// TIA Portal V18 export
// export: Created 2025-12-01T12:38:16.9632914Z, ExportSetting None, DisplayName Totally Integrated Automation Portal, DisplayVersion V18 Update 5, DisplayName TIA Portal Openness, DisplayVersion V18 Update 5, DisplayName TIA Portal Teamcenter Gateway, DisplayVersion V18, DisplayName TIA Portal Version Control Interface, DisplayVersion V18, DisplayName STEP 7 Professional, DisplayVersion V18 Update 5, DisplayName STEP 7 Safety, DisplayVersion V18, DisplayName WinCC Professional, DisplayVersion V18 Update 5
FUNCTION_BLOCK "ST10_Flow15_FRobot_3"   // FB1085, GRAPH
// stored: AcknowledgeErrorsRequired false, AutoNumber false, GraphVersion 6.0, InitialValuesAcquisition false, SetENOAutomatically false
   // inherited from GRAPH_BASE
   VAR_INPUT
      iSysInface : "RCS_SysComInterface_V1";
   END_VAR
   VAR_IN_OUT
      ioPM_Inface : "RCS_PMInterface_V1";
      ioStatus : Int;
   END_VAR
   VAR
      sCtrlMode { S7_SetPoint := 'True'} : "SysFlowCtrlGraph";
      sUpdMES_Data : Bool;   // 更新MES数据
      工件放行中 : Bool;
      前站站号 { ExternalAccessible := 'False'; ExternalVisible := 'False'; ExternalWritable := 'False'} : UInt;
      本站站号 { ExternalAccessible := 'False'; ExternalVisible := 'False'; ExternalWritable := 'False'} : UInt;
      弹窗Temp : Array[1..10] of Int;
      AlarmID : Int;
      TON { S7_SetPoint := 'True'} : Array[0..10] of TON_TIME;
      TOF { S7_SetPoint := 'True'} : Array[0..10] of TOF_TIME;
      sUP { S7_SetPoint := 'True'} : Array[0..10] of Bool;
      更新RFID完成 : Bool;
   END_VAR
   VAR_TEMP
      Tempresult : USInt;
      本站站号乘10 : UInt;
   END_VAR
   // // TON[0] : 托盘流入1托盘到位传感器
   // // TON[1] : 托盘流入1托盘到位传感器
   // // TON[2] : 托盘流入1产品有无传感器
   // // TON[3] : 托盘流入1产品有无传感器
   // // TON[4] : 托盘流入1姿态检测光电2
   // // TON[5] : 托盘流入1姿态检测光电3
   // // TON[0].Q : 托盘流入1托盘到位
   // // TON[1].Q : 托盘流入1托盘无
   // // TON[2].Q : 托盘流入1有产品
   // // TON[3].Q : 托盘流入1无产品
   // // TON[4].Q : 托盘流入1姿态检测光电2
   // // TON[5].Q : 托盘流入1姿态检测光电3
BEGIN
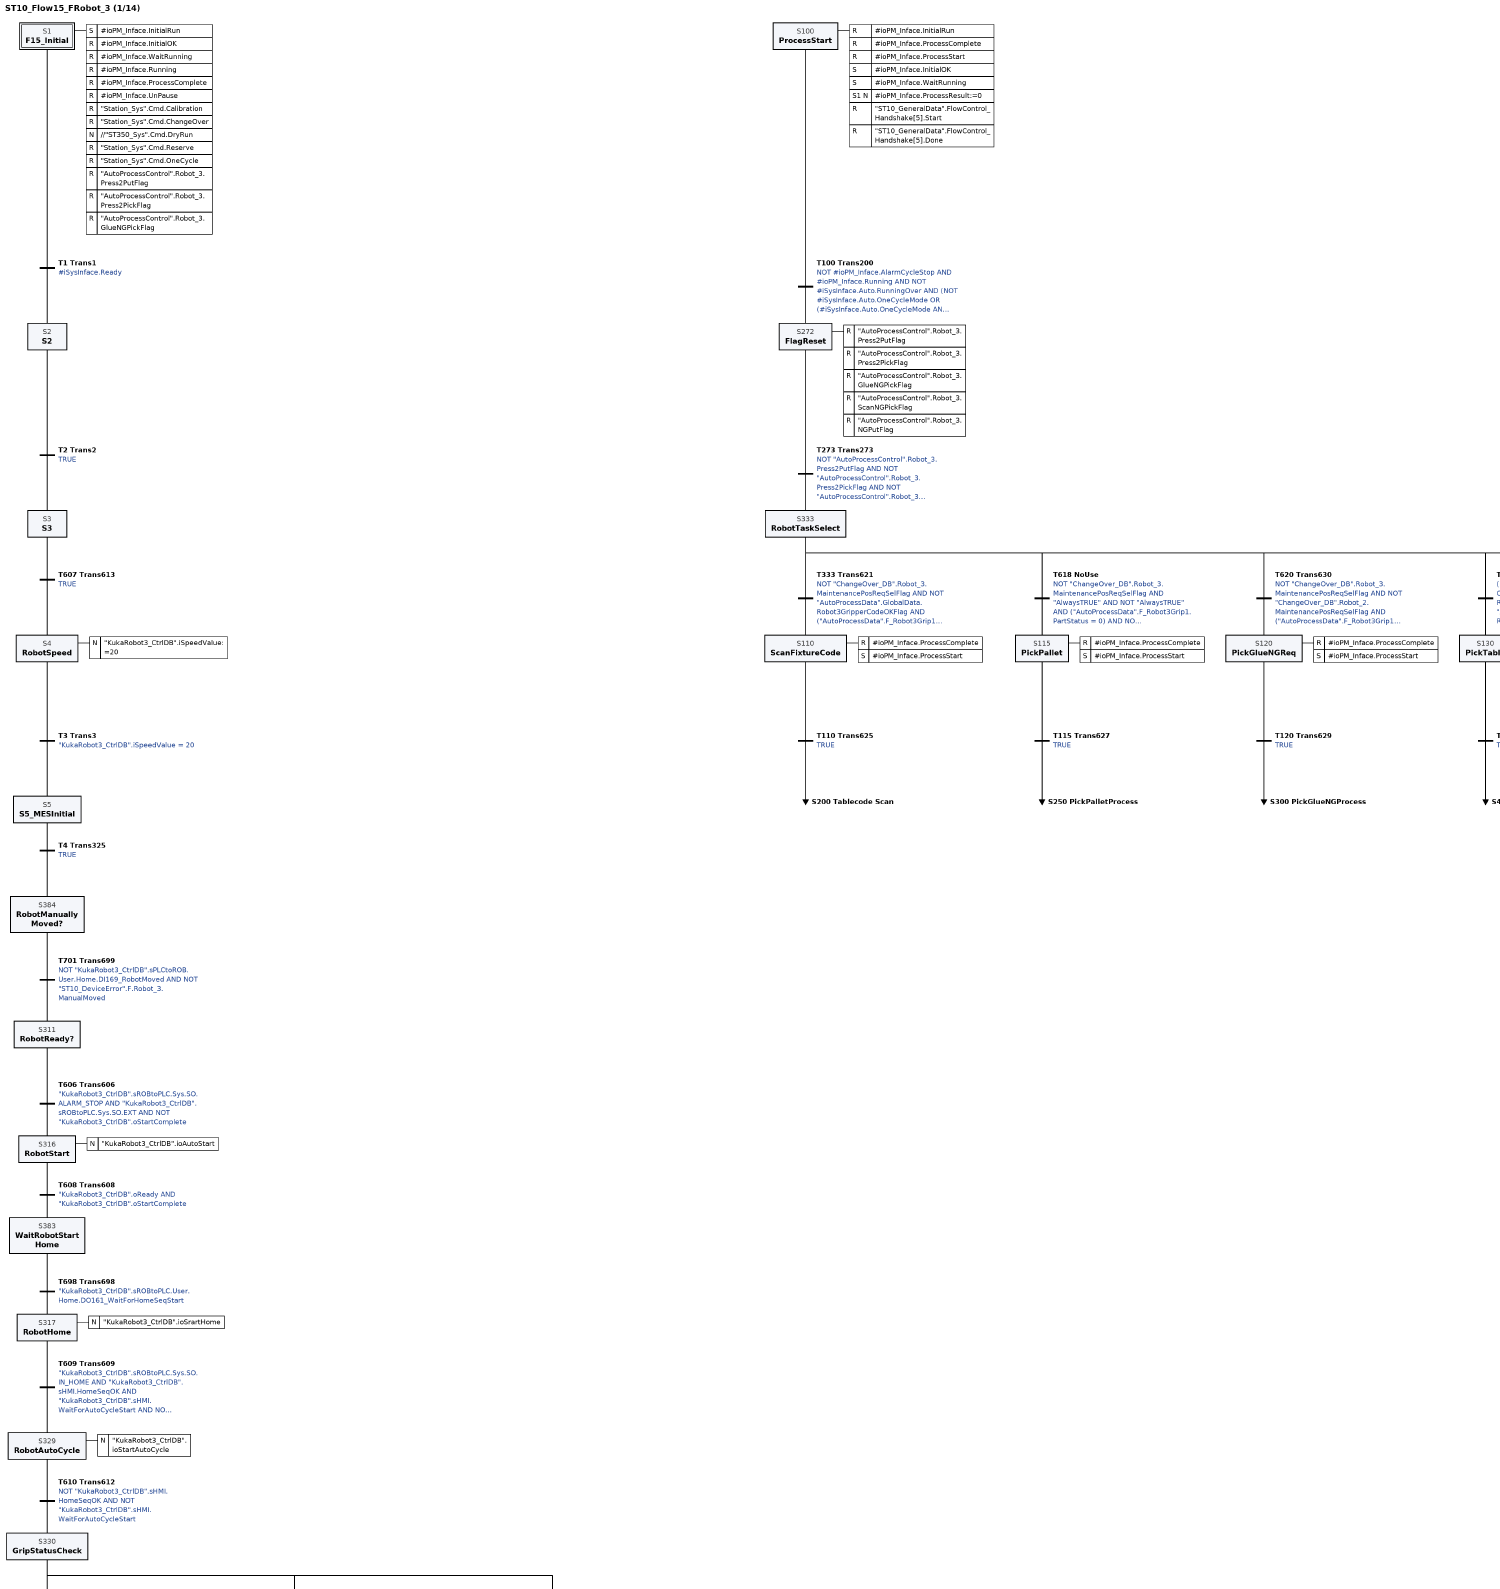
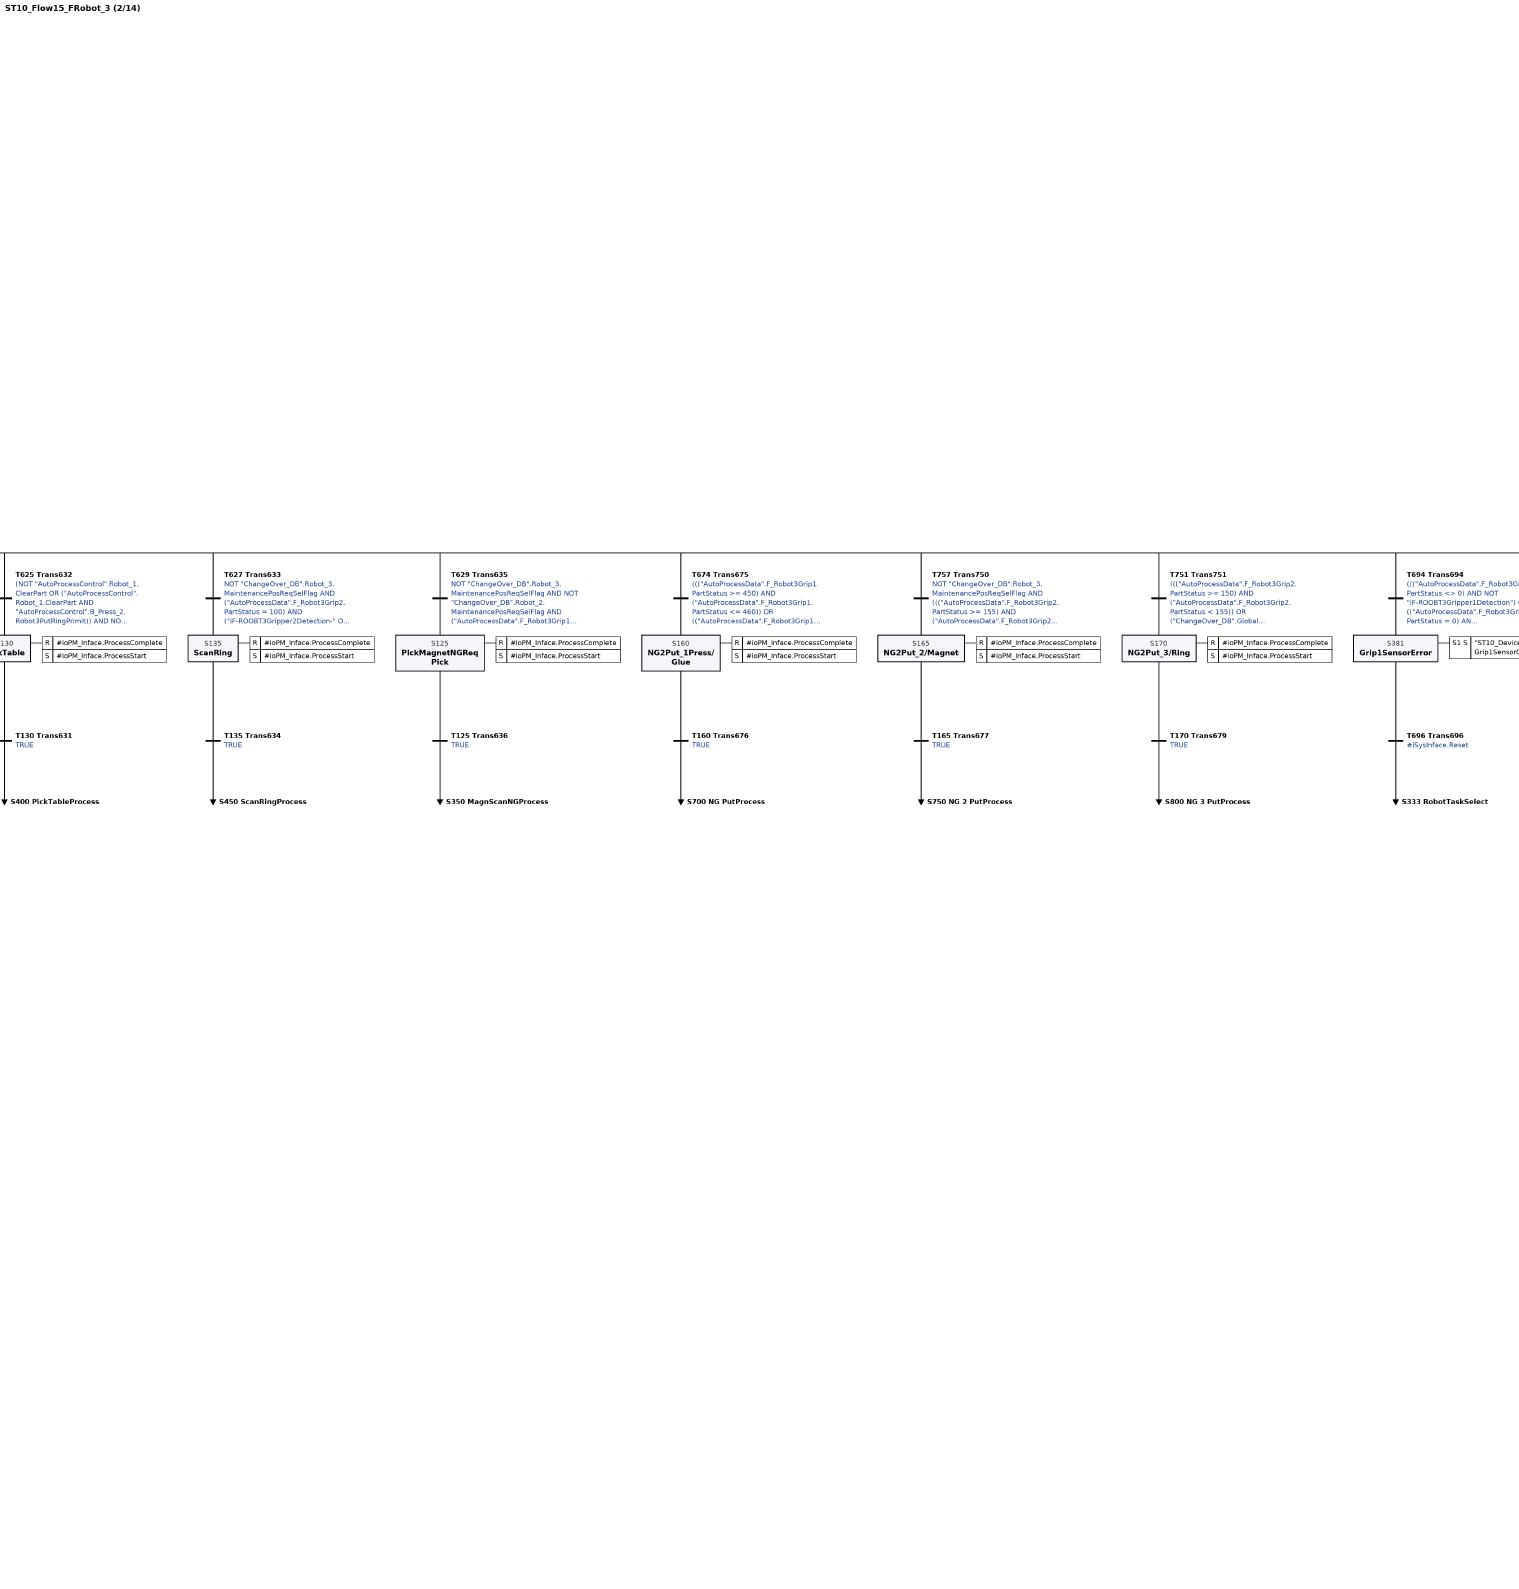
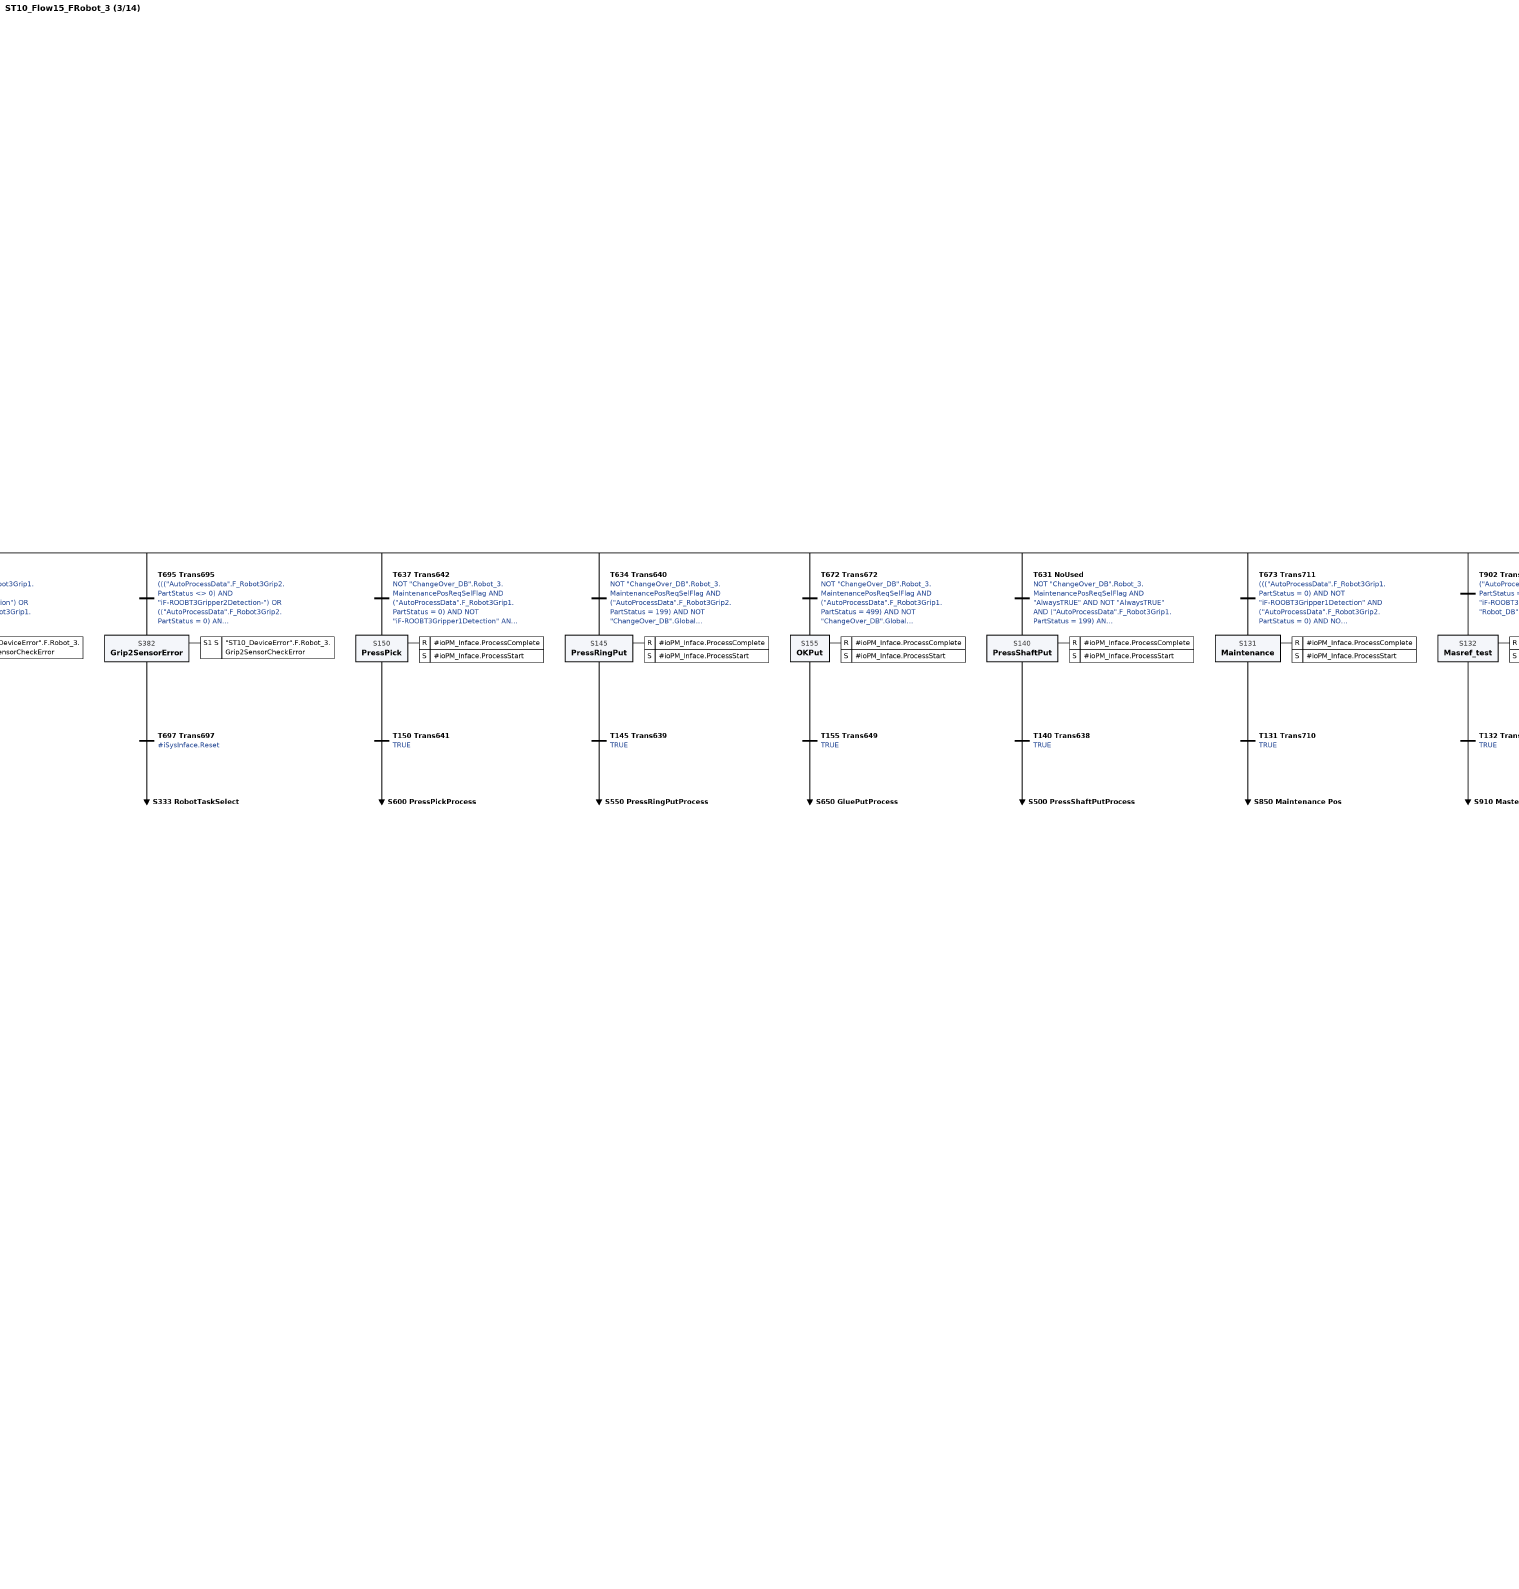
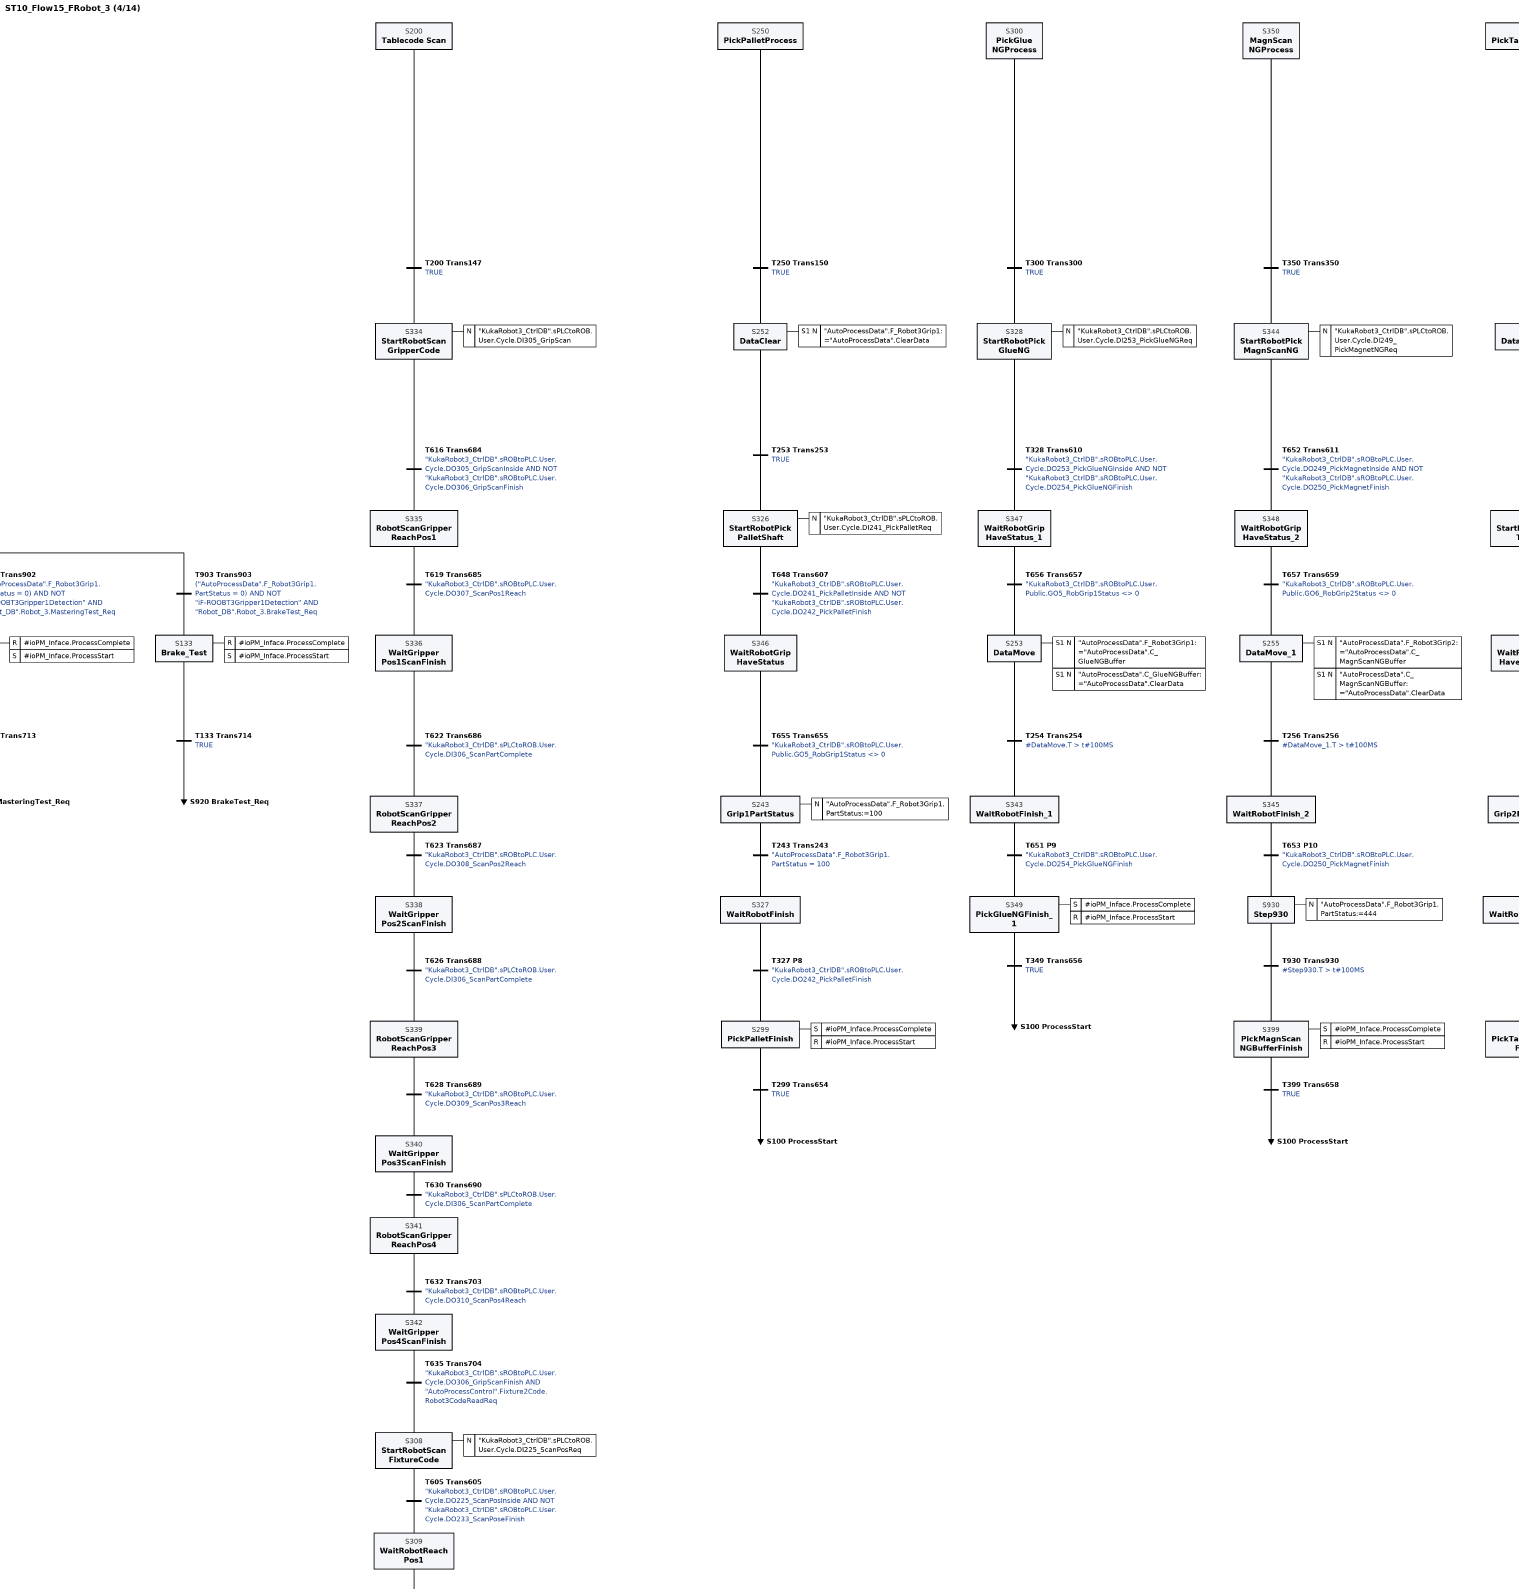
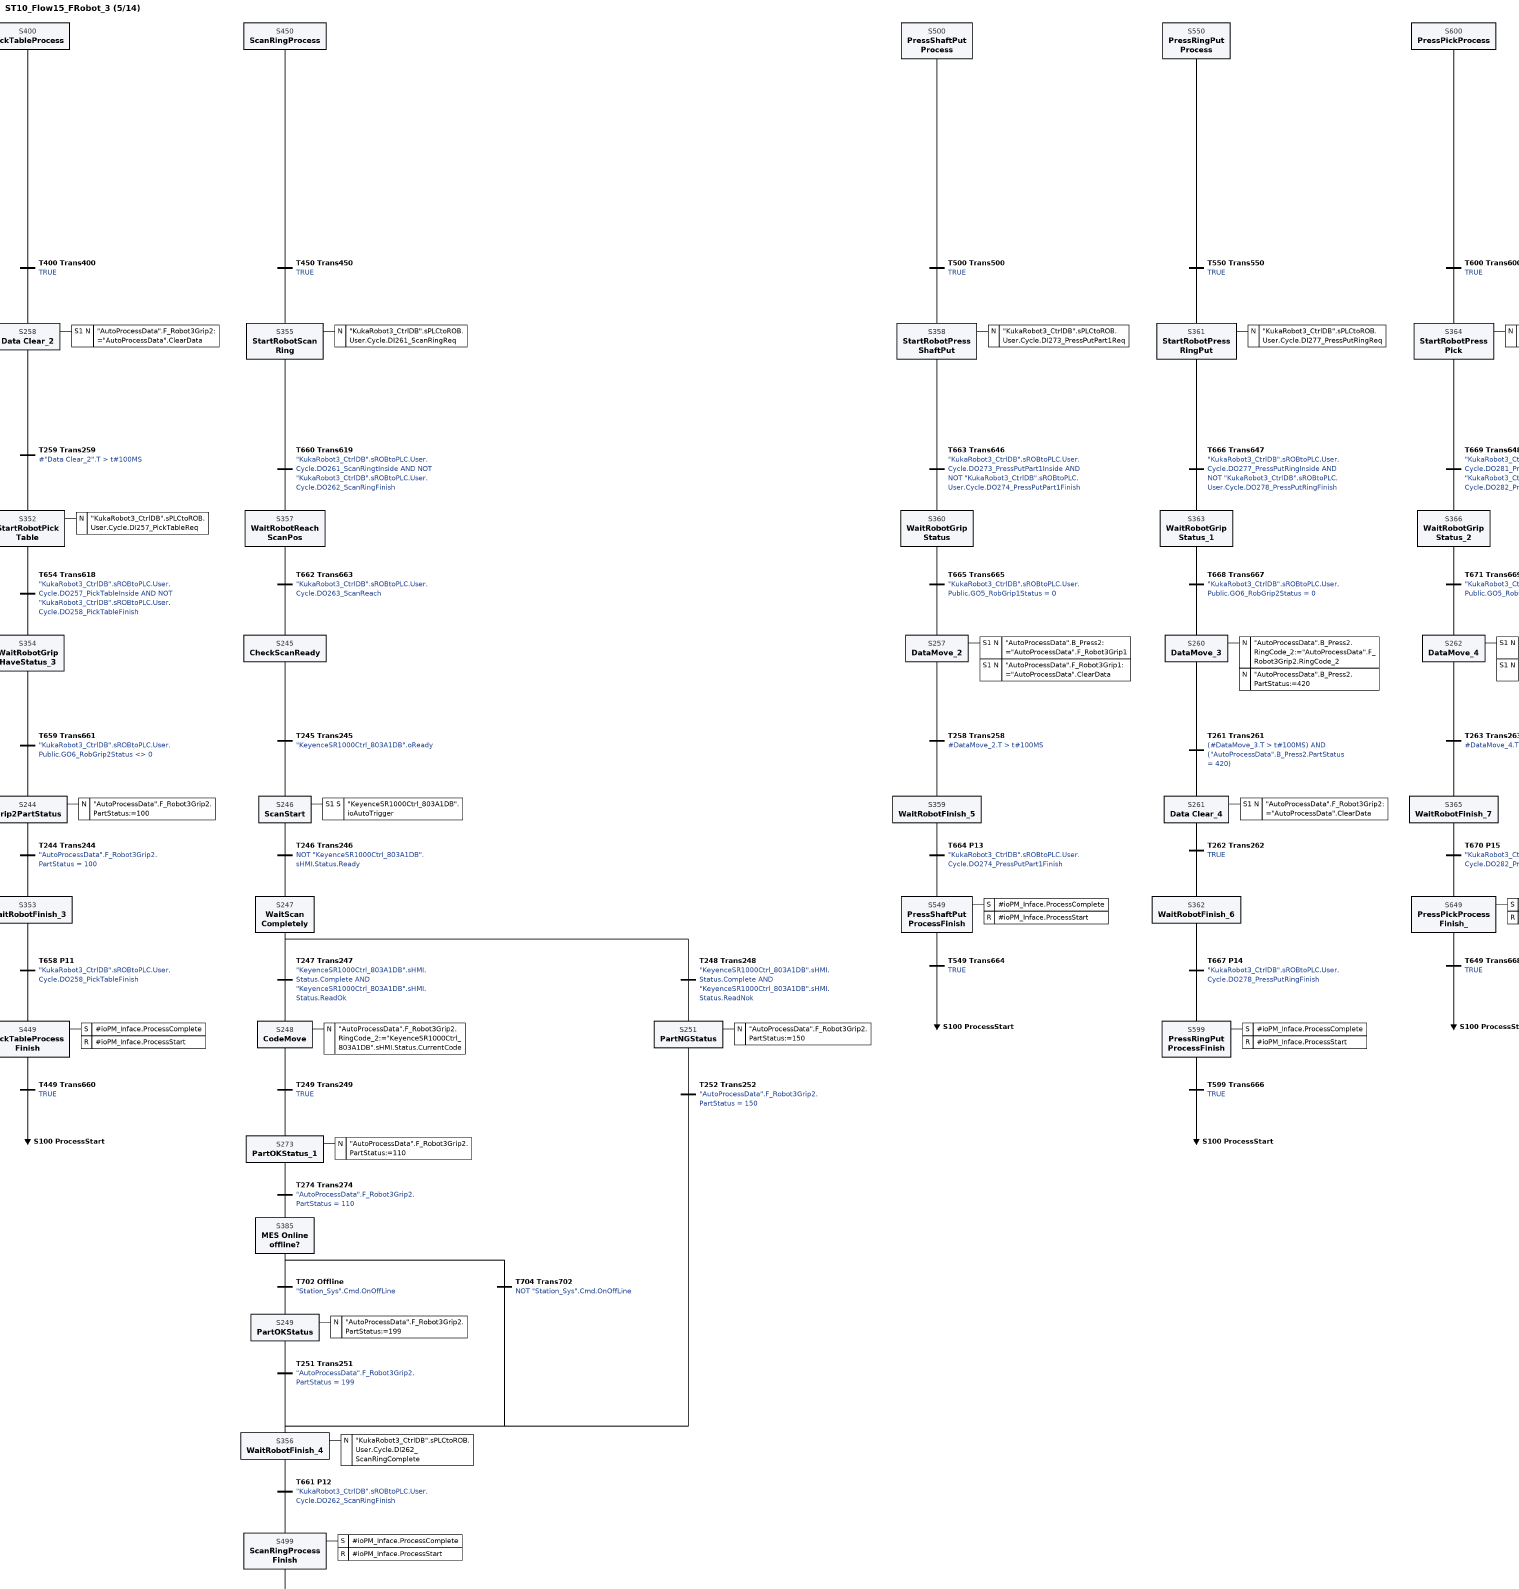
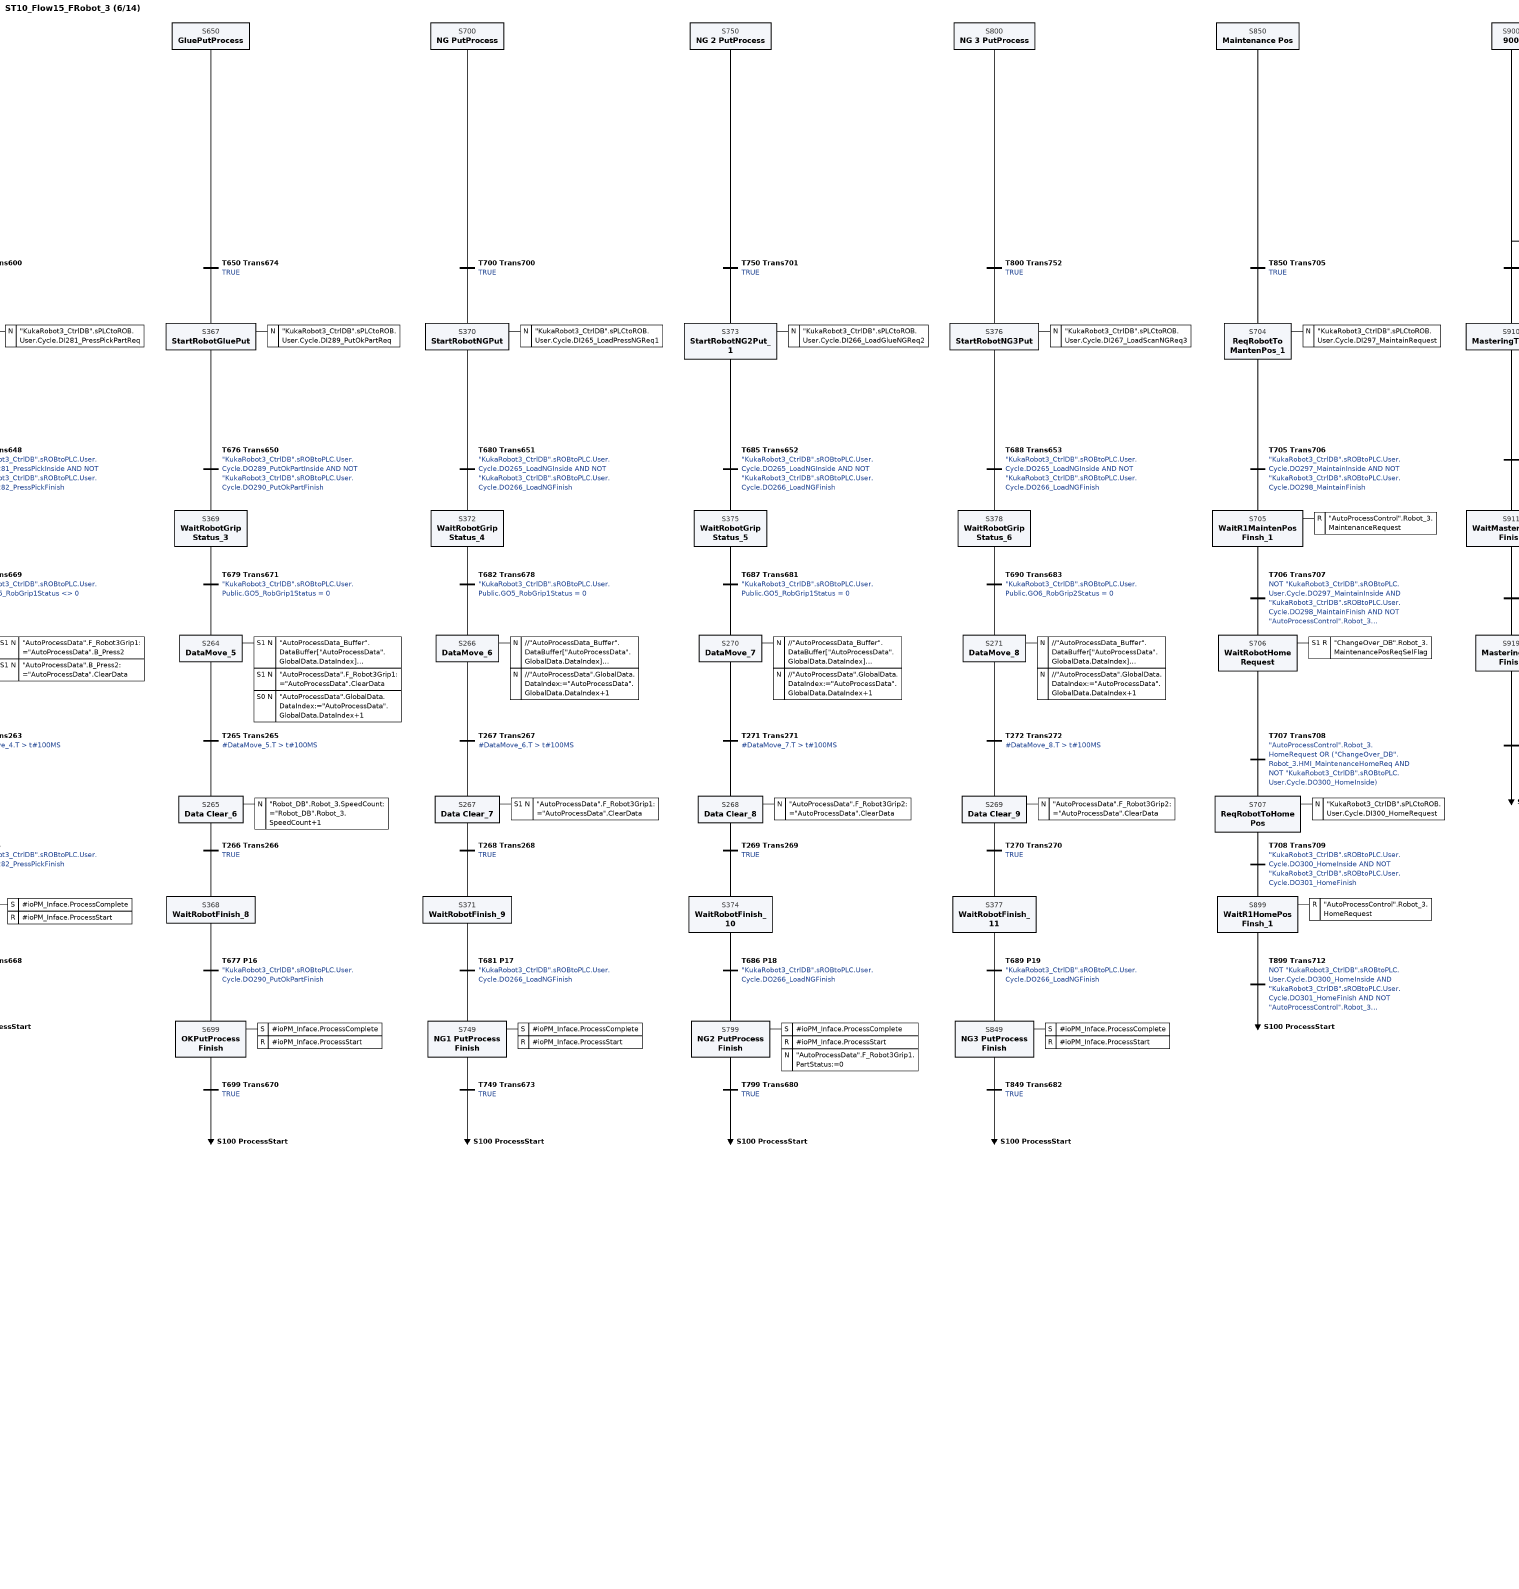
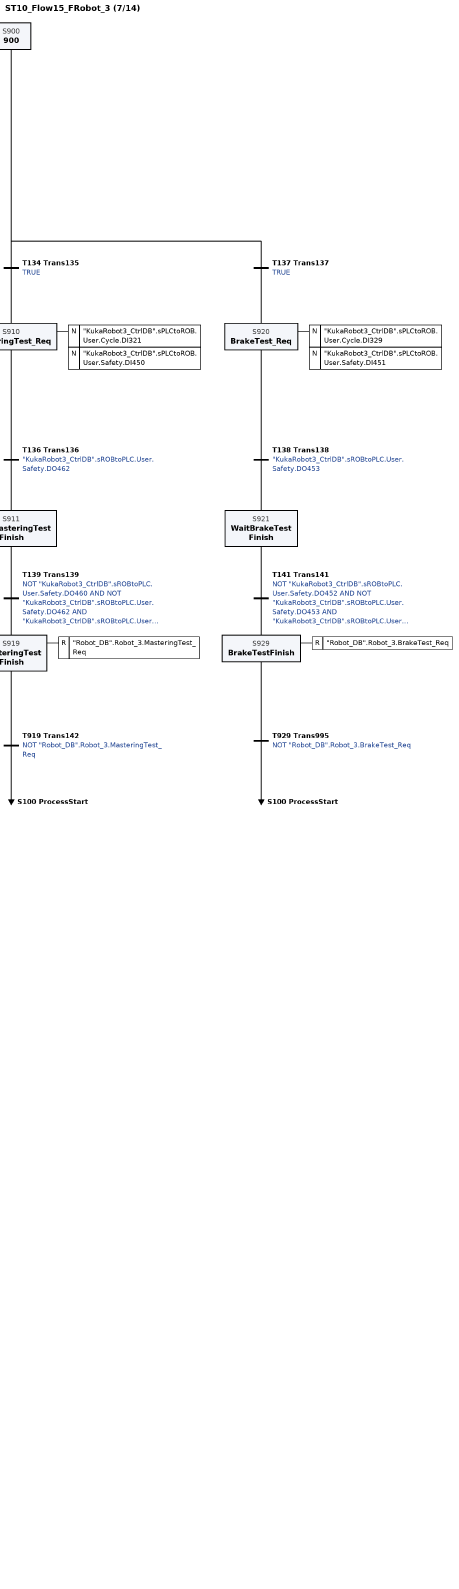
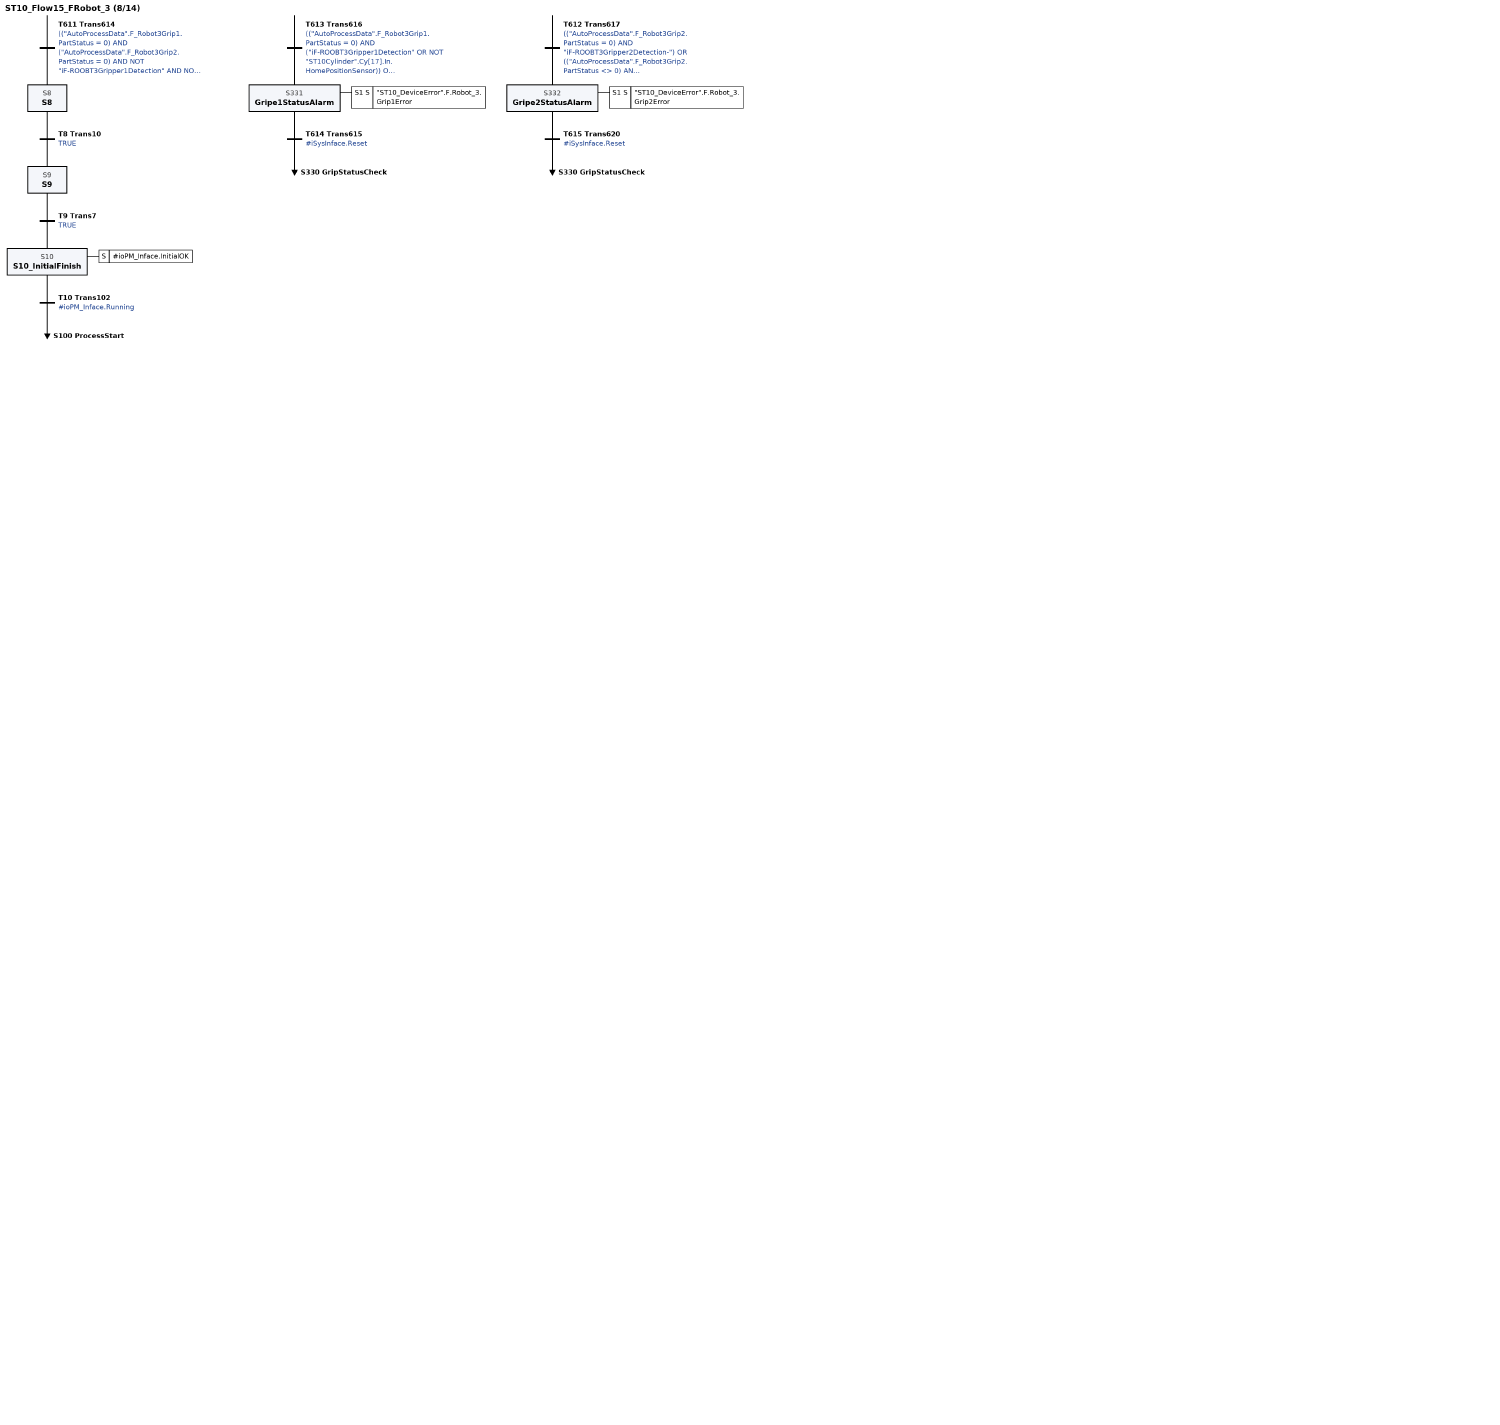
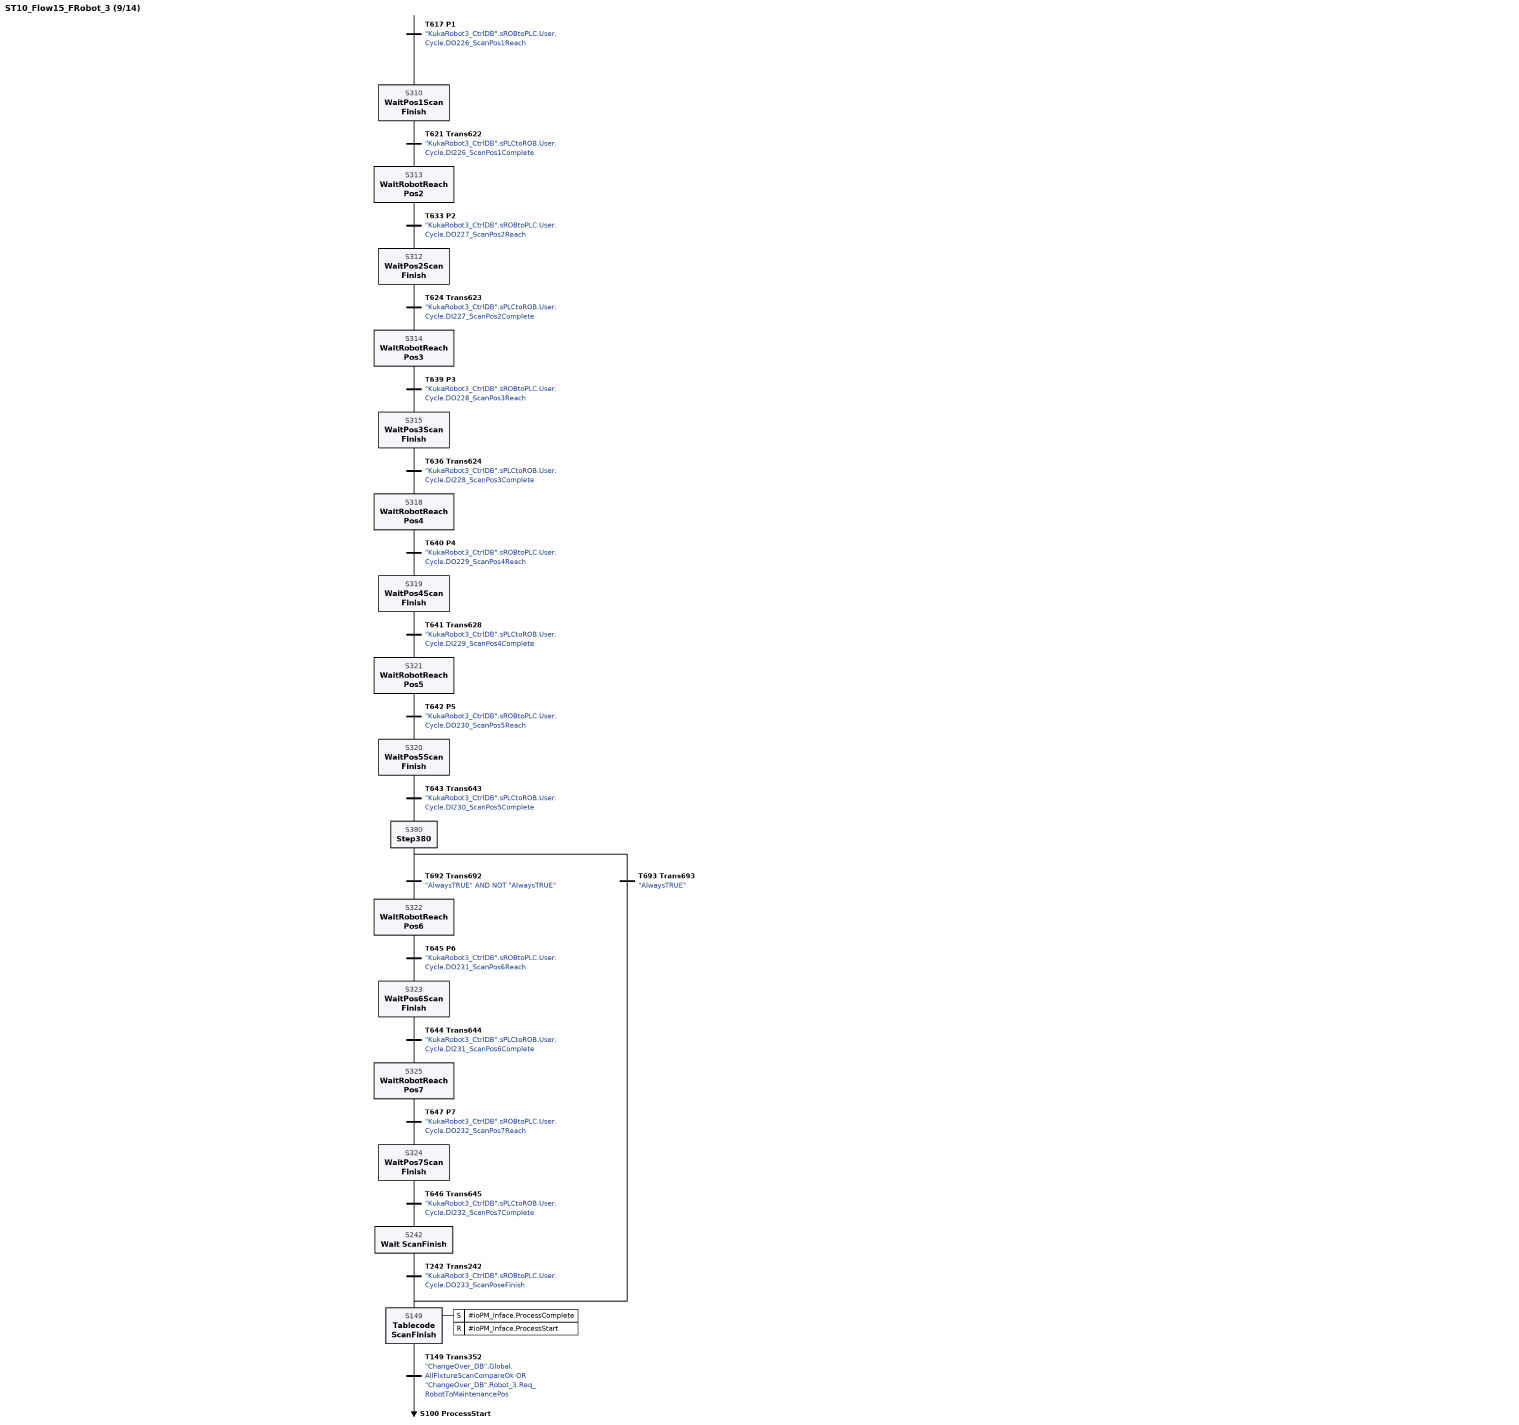
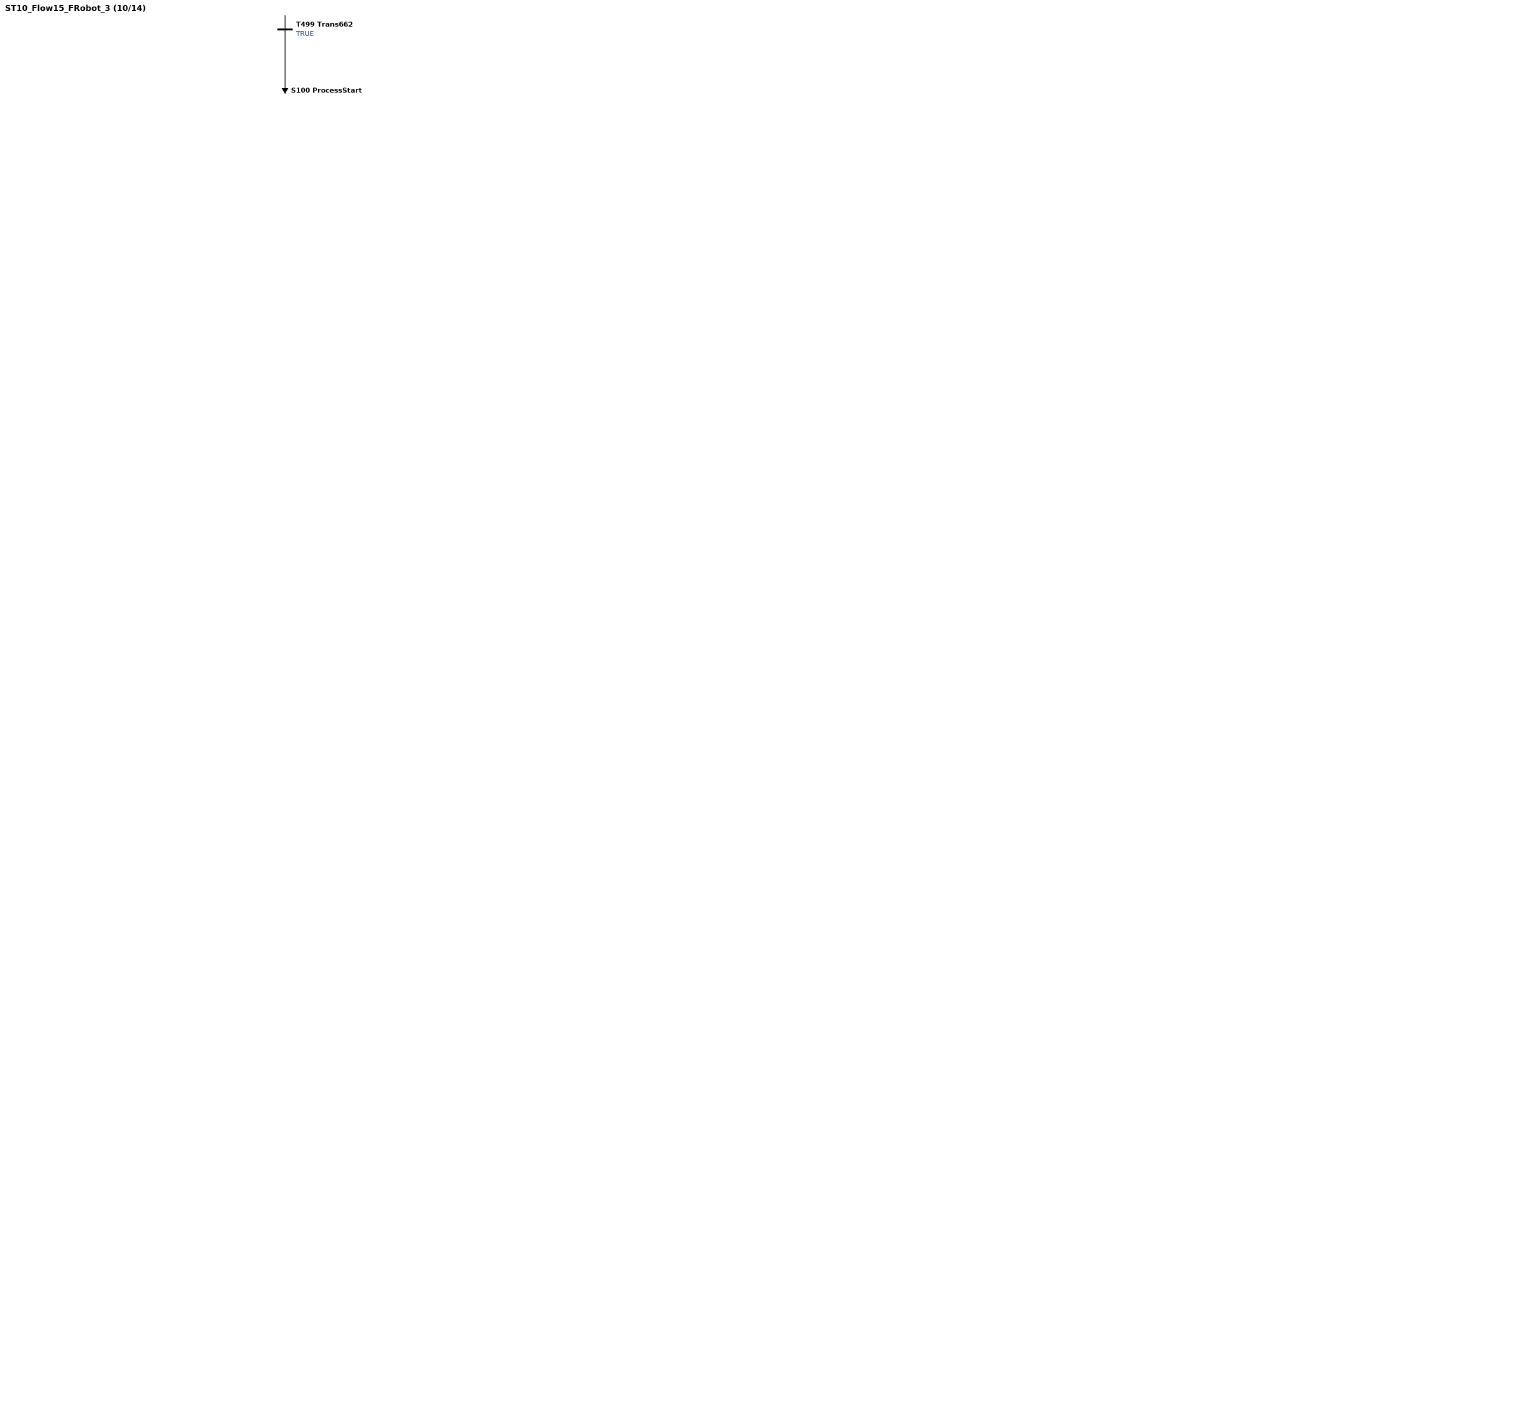
   // permanent pre-instructions
   NETWORK 1
      #TON[10].TON(IN := "AlwaysTRUE" AND "Station_Sys".Alarm.ImmediatelyStop, PT := T#300ms);
      #ioPM_Inface.AlarmImdilyStop := #TON[10].Q;
      #ioPM_Inface.AlarmCycleStop := "AlwaysTRUE" AND "Station_Sys".Alarm.CycleStop;
   NETWORK 2
      IF NOT False THEN
          #sCtrlMode(iSysInface := #iSysInface, ioPM_Inface := #ioPM_Inface, ioGraphCtrl := #RT_DATA.MOP);   // "SysFlowCtrlGraph"
      END_IF;
   NETWORK 3
      #TON[0].TON(IN := "AlwaysTRUE" AND "iA-Rotating product Check", PT := t#500ms);   // 工位11有托盘
      #TON[1].TOF(IN := "AlwaysTRUE" AND NOT "iA-Rotating product Check", PT := T#300ms);   // 工位无托盘
      #TON[2].TON(IN := "AlwaysTRUE", PT := T#300ms);
      #TON[3].TON(IN := "AlwaysTRUE", PT := T#300ms);
      #TON[4].TON(IN := "AlwaysTRUE", PT := T#300ms);
      #TON[5].TON(IN := "AlwaysTRUE", PT := T#300ms);
   NETWORK 4
      #前站站号 := 345;
      #本站站号 := 350;

   // sequencer 1: S01-S99 初始化 / S01-S99 Initial
   INITIAL_STEP F15_Initial:   // S1, max time T#10S, warning time T#7S
              S    #ioPM_Inface.InitialRun
              R    #ioPM_Inface.InitialOK
              R    #ioPM_Inface.WaitRunning
              R    #ioPM_Inface.Running
              R    #ioPM_Inface.ProcessComplete
              R    #ioPM_Inface.UnPause
              R    "Station_Sys".Cmd.Calibration
              R    "Station_Sys".Cmd.ChangeOver
                   //"ST350_Sys".Cmd.DryRun
              R    "Station_Sys".Cmd.Reserve
              R    "Station_Sys".Cmd.OneCycle
              R    "AutoProcessControl".Robot_3.Press2PutFlag
              R    "AutoProcessControl".Robot_3.Press2PickFlag
              R    "AutoProcessControl".Robot_3.GlueNGPickFlag
              R    "AutoProcessControl".Robot_3.ScanNGPickFlag
              R    "AutoProcessControl".Robot_3.NGPutFlag
              R    #ioPM_Inface.ProcessStart
          S1  R    "ChangeOver_DB".Robot_3.MaintenancePosReqSelFlag
                   //"Robot_DB".Robot_3.MasteringTest_Req
                   //"Robot_DB".Robot_3.BrakeTest_Req
   END_STEP
   TRANSITION Trans1 FROM F15_Initial TO S2   // T1
      := #iSysInface.Ready;
   END_TRANSITION
   STEP S2:   // S2, max time T#10S, warning time T#7S
   END_STEP
   TRANSITION Trans2 FROM S2 TO S3   // T2
      := TRUE;
   END_TRANSITION
   STEP RobotSpeed:   // S4, max time T#10S, warning time T#7S
              N    "KukaRobot3_CtrlDB".iSpeedValue:=20
   END_STEP
   TRANSITION Trans3 FROM RobotSpeed TO S5_MESInitial   // T3
      := "KukaRobot3_CtrlDB".iSpeedValue = 20;
   END_TRANSITION
   STEP S5_MESInitial:   // S5, max time T#10S, warning time T#7S
   END_STEP
   TRANSITION Trans325 FROM S5_MESInitial TO "RobotManuallyMoved?"   // T4
      := TRUE;
   END_TRANSITION
   STEP S10_InitialFinish:   // S10, max time T#10S, warning time T#7S
              S    #ioPM_Inface.InitialOK
   END_STEP
   TRANSITION Trans102 FROM S10_InitialFinish TO ProcessStart   // T10, jump
      := #ioPM_Inface.Running;
   END_TRANSITION
   STEP S3:   // S3, max time T#10S, warning time T#7S
   END_STEP
   TRANSITION Trans613 FROM S3 TO RobotSpeed   // T607
      := TRUE;
   END_TRANSITION
   STEP S8:   // S8, max time T#10S, warning time T#7S
   END_STEP
   TRANSITION Trans10 FROM S8 TO S9   // T8
      := TRUE;
   END_TRANSITION
   STEP S9:   // S9, max time T#10S, warning time T#7S
   END_STEP
   TRANSITION Trans7 FROM S9 TO S10_InitialFinish   // T9
      := TRUE;
   END_TRANSITION
   STEP "RobotReady?":   // S311, max time T#10S, warning time T#7S
   END_STEP
   TRANSITION Trans606 FROM "RobotReady?" TO RobotStart   // T606
      := "KukaRobot3_CtrlDB".sROBtoPLC.Sys.SO.ALARM_STOP AND "KukaRobot3_CtrlDB".sROBtoPLC.Sys.SO.EXT AND NOT "KukaRobot3_CtrlDB".oStartComplete;
   END_TRANSITION
   STEP RobotStart:   // S316, max time T#10S, warning time T#7S
              N    "KukaRobot3_CtrlDB".ioAutoStart
   END_STEP
   TRANSITION Trans608 FROM RobotStart TO WaitRobotStartHome   // T608
      := "KukaRobot3_CtrlDB".oReady AND "KukaRobot3_CtrlDB".oStartComplete;
   END_TRANSITION
   STEP RobotHome:   // S317, max time T#10S, warning time T#7S
              N    "KukaRobot3_CtrlDB".ioSrartHome
   END_STEP
   TRANSITION Trans609 FROM RobotHome TO RobotAutoCycle   // T609
      := "KukaRobot3_CtrlDB".sROBtoPLC.Sys.SO.IN_HOME AND "KukaRobot3_CtrlDB".sHMI.HomeSeqOK AND "KukaRobot3_CtrlDB".sHMI.WaitForAutoCycleStart AND NOT "KukaRobot3_CtrlDB".sHMI.GoHomeFail;
   END_TRANSITION
   STEP RobotAutoCycle:   // S329, max time T#10S, warning time T#7S
              N    "KukaRobot3_CtrlDB".ioStartAutoCycle
   END_STEP
   TRANSITION Trans612 FROM RobotAutoCycle TO GripStatusCheck   // T610
      := NOT "KukaRobot3_CtrlDB".sHMI.HomeSeqOK AND NOT "KukaRobot3_CtrlDB".sHMI.WaitForAutoCycleStart;
   END_TRANSITION
   STEP GripStatusCheck:   // S330, max time T#10S, warning time T#7S
   END_STEP
   TRANSITION Trans614 FROM GripStatusCheck TO S8   // T611
      := (("AutoProcessData".F_Robot3Grip1.PartStatus = 0) AND ("AutoProcessData".F_Robot3Grip2.PartStatus = 0) AND NOT "iF-ROOBT3Gripper1Detection" AND NOT "iF-ROOBT3Gripper2Detection-") OR (("AutoProcessData".F_Robot3Grip1.PartStatus <> 0) AND NOT "ST10Cylinder".Cy[17].In.WorkPositionSensor AND NOT "ST10Cylinder".Cy[17].In.HomePositionSensor) OR (("AutoProcessData".F_Robot3Grip2.PartStatus <> 0) AND NOT "iF-ROOBT3Gripper2Detection-" AND NOT "ST10Cylinder".Cy[18].In.HomePositionSensor);
   END_TRANSITION
   TRANSITION Trans616 FROM GripStatusCheck TO Gripe1StatusAlarm   // T613
      := (("AutoProcessData".F_Robot3Grip1.PartStatus = 0) AND ("iF-ROOBT3Gripper1Detection" OR NOT "ST10Cylinder".Cy[17].In.HomePositionSensor)) OR (("AutoProcessData".F_Robot3Grip1.PartStatus <> 0) AND (NOT "iF-ROOBT3Gripper1Detection" OR "ST10Cylinder".Cy[17].In.HomePositionSensor));
   END_TRANSITION
   TRANSITION Trans617 FROM GripStatusCheck TO Gripe2StatusAlarm   // T612
      := (("AutoProcessData".F_Robot3Grip2.PartStatus = 0) AND "iF-ROOBT3Gripper2Detection-") OR (("AutoProcessData".F_Robot3Grip2.PartStatus <> 0) AND "iF-ROOBT3Gripper2Detection-");
   END_TRANSITION
   STEP Gripe1StatusAlarm:   // S331, max time T#10S, warning time T#7S
          S1  S    "ST10_DeviceError".F.Robot_3.Grip1Error
   END_STEP
   TRANSITION Trans615 FROM Gripe1StatusAlarm TO GripStatusCheck   // T614, jump
      := #iSysInface.Reset;
   END_TRANSITION
   STEP Gripe2StatusAlarm:   // S332, max time T#10S, warning time T#7S
          S1  S    "ST10_DeviceError".F.Robot_3.Grip2Error
   END_STEP
   TRANSITION Trans620 FROM Gripe2StatusAlarm TO GripStatusCheck   // T615, jump
      := #iSysInface.Reset;
   END_TRANSITION
   STEP WaitRobotStartHome:   // S383, max time T#10S, warning time T#7S
   END_STEP
   TRANSITION Trans698 FROM WaitRobotStartHome TO RobotHome   // T698
      := "KukaRobot3_CtrlDB".sROBtoPLC.User.Home.DO161_WaitForHomeSeqStart;
   END_TRANSITION
   STEP "RobotManuallyMoved?":   // S384, max time T#10S, warning time T#7S
   END_STEP
   TRANSITION Trans699 FROM "RobotManuallyMoved?" TO "RobotReady?"   // T701
      := NOT "KukaRobot3_CtrlDB".sPLCtoROB.User.Home.DI169_RobotMoved AND NOT "ST10_DeviceError".F.Robot_3.ManualMoved;
   END_TRANSITION

   // sequencer 2: S100-S199 等待到位 / S100-S199 RobotTask
   STEP ProcessStart:   // S100, max time T#10S, warning time T#7S
      // 自动等待开始运行
              R    #ioPM_Inface.InitialRun
              R    #ioPM_Inface.ProcessComplete
              R    #ioPM_Inface.ProcessStart
              S    #ioPM_Inface.InitialOK
              S    #ioPM_Inface.WaitRunning
          S1  N    #ioPM_Inface.ProcessResult:=0
              R    "ST10_GeneralData".FlowControl_Handshake[5].Start
              R    "ST10_GeneralData".FlowControl_Handshake[5].Done
   END_STEP
   TRANSITION Trans200 FROM ProcessStart TO FlagReset   // T100
      := NOT #ioPM_Inface.AlarmCycleStop AND #ioPM_Inface.Running AND NOT #iSysInface.Auto.RunningOver AND (NOT #iSysInface.Auto.OneCycleMode OR (#iSysInface.Auto.OneCycleMode AND #ioPM_Inface.TriggerOneCycle));
   END_TRANSITION
   STEP PressShaftPut:   // S140, max time T#10S, warning time T#7S
              R    #ioPM_Inface.ProcessComplete
              S    #ioPM_Inface.ProcessStart
   END_STEP
   TRANSITION Trans638 FROM PressShaftPut TO PressShaftPutProcess   // T140, jump
      := TRUE;
   END_TRANSITION
   STEP ScanFixtureCode:   // S110, max time T#10S, warning time T#7S
              R    #ioPM_Inface.ProcessComplete
              S    #ioPM_Inface.ProcessStart
   END_STEP
   TRANSITION Trans625 FROM ScanFixtureCode TO "Tablecode Scan"   // T110, jump
      := TRUE;
   END_TRANSITION
   STEP RobotTaskSelect:   // S333, max time T#10S, warning time T#7S
   END_STEP
   TRANSITION Trans621 FROM RobotTaskSelect TO ScanFixtureCode   // T333
      := NOT "ChangeOver_DB".Robot_3.MaintenancePosReqSelFlag AND NOT "AutoProcessData".GlobalData.Robot3GripperCodeOKFlag AND ("AutoProcessData".F_Robot3Grip1.PartStatus = 0) AND NOT "iF-ROOBT3Gripper1Detection" AND NOT "KukaRobot2_CtrlDB".sROBtoPLC.User.Cycle.DO253_GlueNGPutInside AND NOT "KukaRobot2_CtrlDB".sROBtoPLC.User.Cycle.DO249_ScanNGPutInside AND NOT "KukaRobot2_CtrlDB".sROBtoPLC.User.Cycle.DO273_PressPutPart1Inside AND NOT "PalletNGData".UnLoadingNGPallet.OpenFlag AND "AutoProcessControl".Robot_3.GripScanRequest AND NOT "Robot_DB".Robot_3.MasteringTest_Req AND NOT "Robot_DB".Robot_3.BrakeTest_Req;
   END_TRANSITION
   TRANSITION NoUse FROM RobotTaskSelect TO PickPallet   // T618
      := NOT "ChangeOver_DB".Robot_3.MaintenancePosReqSelFlag AND "AlwaysTRUE" AND NOT "AlwaysTRUE" AND ("AutoProcessData".F_Robot3Grip1.PartStatus = 0) AND NOT "iF-ROOBT3Gripper1Detection" AND "ST10Cylinder".Cy[17].In.HomePositionSensor AND "AutoProcessControl".H_ShafeLine.Robot1PickPrimit AND NOT "PalletNGData".UnLoadingNGPallet.OpenFlag AND "AutoProcessControl".A_ScanRotary.Robot1PutPrimit AND NOT "Robot_DB".Robot_3.MasteringTest_Req AND NOT "Robot_DB".Robot_3.BrakeTest_Req;
   END_TRANSITION
   TRANSITION Trans630 FROM RobotTaskSelect TO PickGlueNGReq   // T620
      := NOT "ChangeOver_DB".Robot_3.MaintenancePosReqSelFlag AND NOT "ChangeOver_DB".Robot_2.MaintenancePosReqSelFlag AND ("AutoProcessData".F_Robot3Grip1.PartStatus = 0) AND NOT "iF-ROOBT3Gripper1Detection" AND "iE-NG-03ShaftDispenseNGDetection" AND "KukaRobot2_CtrlDB".sROBtoPLC.User.Home.DO181_Robot3Area AND NOT "KukaRobot2_CtrlDB".sROBtoPLC.User.Cycle.DO253_GlueNGPutInside AND NOT "KukaRobot2_CtrlDB".sROBtoPLC.User.Cycle.DO249_ScanNGPutInside AND NOT "KukaRobot2_CtrlDB".sROBtoPLC.User.Cycle.DO273_PressPutPart1Inside AND NOT "AutoProcessControl".Robot_2.GlueNGPutFlag AND NOT "AutoProcessControl".Robot_2.ScanNGPutFlag AND NOT "AutoProcessControl".Robot_2.Press2PutFlag AND NOT "PalletNGData".UnLoadingNGPallet.OpenFlag AND "AutoProcessControl".NGBuffer.PickGlueNGPrimit AND NOT "Robot_DB".Robot_3.MasteringTest_Req AND NOT "Robot_DB".Robot_3.BrakeTest_Req;
   END_TRANSITION
   TRANSITION Trans632 FROM RobotTaskSelect TO PickTable   // T625
      := (NOT "AutoProcessControl".Robot_1.ClearPart OR ("AutoProcessControl".Robot_1.ClearPart AND "AutoProcessControl".B_Press_2.Robot3PutRingPrimit)) AND NOT "ChangeOver_DB".Robot_3.MaintenancePosReqSelFlag AND ("AutoProcessData".F_Robot3Grip1.PartStatus = 0) AND NOT "iF-ROOBT3Gripper1Detection" AND ("AutoProcessData".F_Robot3Grip2.PartStatus = 0) AND NOT "iF-ROOBT3Gripper2Detection-" AND NOT "iE-NG-03MagnetDispenseNGDetection" AND NOT "iE-NG-03ShaftDispenseNGDetection" AND NOT "PalletNGData".UnLoadingNGPallet.OpenFlag AND "AutoProcessControl".A_Table_2Loading.Robot3PickPrimit AND NOT "Robot_DB".Robot_3.MasteringTest_Req AND NOT "Robot_DB".Robot_3.BrakeTest_Req;
   END_TRANSITION
   TRANSITION Trans633 FROM RobotTaskSelect TO ScanRing   // T627
      := NOT "ChangeOver_DB".Robot_3.MaintenancePosReqSelFlag AND ("AutoProcessData".F_Robot3Grip2.PartStatus = 100) AND ("iF-ROOBT3Gripper2Detection-" OR "AlwaysTRUE") AND NOT "ChangeOver_DB".Global.ManualModeFlag AND NOT "PalletNGData".UnLoadingNGPallet.OpenFlag AND NOT "ST10Cylinder".Cy[18].In.HomePositionSensor AND NOT "Robot_DB".Robot_3.MasteringTest_Req AND NOT "Robot_DB".Robot_3.BrakeTest_Req;
   END_TRANSITION
   TRANSITION Trans635 FROM RobotTaskSelect TO PickMagnetNGReqPick   // T629
      := NOT "ChangeOver_DB".Robot_3.MaintenancePosReqSelFlag AND NOT "ChangeOver_DB".Robot_2.MaintenancePosReqSelFlag AND ("AutoProcessData".F_Robot3Grip1.PartStatus = 0) AND NOT "iF-ROOBT3Gripper1Detection" AND ("AutoProcessData".F_Robot3Grip2.PartStatus = 0) AND NOT "iF-ROOBT3Gripper2Detection-" AND "iE-NG-03MagnetDispenseNGDetection" AND "KukaRobot2_CtrlDB".sROBtoPLC.User.Home.DO181_Robot3Area AND NOT "KukaRobot2_CtrlDB".sROBtoPLC.User.Cycle.DO253_GlueNGPutInside AND NOT "KukaRobot2_CtrlDB".sROBtoPLC.User.Cycle.DO249_ScanNGPutInside AND NOT "KukaRobot2_CtrlDB".sROBtoPLC.User.Cycle.DO273_PressPutPart1Inside AND NOT "AutoProcessControl".Robot_2.GlueNGPutFlag AND NOT "AutoProcessControl".Robot_2.ScanNGPutFlag AND NOT "AutoProcessControl".Robot_2.Press2PutFlag AND NOT "PalletNGData".UnLoadingNGPallet.OpenFlag AND "AutoProcessControl".NGBuffer.Robot3PPickMagnetNGPrimit AND NOT "Robot_DB".Robot_3.MasteringTest_Req AND NOT "Robot_DB".Robot_3.BrakeTest_Req;
   END_TRANSITION
   TRANSITION Trans675 FROM RobotTaskSelect TO "NG2Put_1Press/Glue"   // T674
      := ((("AutoProcessData".F_Robot3Grip1.PartStatus >= 450) AND ("AutoProcessData".F_Robot3Grip1.PartStatus <= 460)) OR (("AutoProcessData".F_Robot3Grip1.PartStatus >= 350) AND ("AutoProcessData".F_Robot3Grip1.PartStatus <= 360))) AND NOT "ChangeOver_DB".Robot_3.MaintenancePosReqSelFlag AND ("iF-ROOBT3Gripper1Detection" OR "AlwaysTRUE") AND NOT "ST10Cylinder".Cy[17].In.HomePositionSensor AND NOT "PalletNGData".UnLoadingNGPallet.OpenFlag AND "AutoProcessControl".NG_2.Robot3PutPrimit_1;
   END_TRANSITION
   TRANSITION Trans750 FROM RobotTaskSelect TO "NG2Put_2/Magnet"   // T757
      := NOT "ChangeOver_DB".Robot_3.MaintenancePosReqSelFlag AND ((("AutoProcessData".F_Robot3Grip2.PartStatus >= 155) AND ("AutoProcessData".F_Robot3Grip2.PartStatus <= 160)) OR ("AutoProcessData".F_Robot3Grip1.PartStatus = 444)) AND ("iF-ROOBT3Gripper2Detection-" OR "AlwaysTRUE") AND NOT "ST10Cylinder".Cy[18].In.HomePositionSensor AND NOT "PalletNGData".UnLoadingNGPallet.OpenFlag AND "AutoProcessControl".NG_2.Robot3PutPrimit_2;
   END_TRANSITION
   TRANSITION Trans751 FROM RobotTaskSelect TO "NG2Put_3/Ring"   // T751
      := ((("AutoProcessData".F_Robot3Grip2.PartStatus >= 150) AND ("AutoProcessData".F_Robot3Grip2.PartStatus < 155)) OR ("ChangeOver_DB".Global.ManualModeFlag AND ("AutoProcessData".F_Robot3Grip2.PartStatus = 100)) OR (("AutoProcessData".F_Robot3Grip2.PartStatus = 199) AND ("AutoProcessData".F_Robot2Grip2.PartStatus = 155) AND ("AutoProcessData".C_MagnScanNGBuffer.PartStatus = 155))) AND NOT "ChangeOver_DB".Robot_3.MaintenancePosReqSelFlag AND ("iF-ROOBT3Gripper2Detection-" OR "AlwaysTRUE") AND NOT "ST10Cylinder".Cy[18].In.HomePositionSensor AND NOT "PalletNGData".UnLoadingNGPallet.OpenFlag AND "AutoProcessControl".NG_2.Robot3PutPrimit_3;
   END_TRANSITION
   TRANSITION Trans694 FROM RobotTaskSelect TO Grip1SensorError   // T694
      := ((("AutoProcessData".F_Robot3Grip1.PartStatus <> 0) AND NOT "iF-ROOBT3Gripper1Detection") OR (("AutoProcessData".F_Robot3Grip1.PartStatus = 0) AND ("iF-ROOBT3Gripper1Detection" OR "AlwaysTRUE"))) AND (#RobotTaskSelect.T > t#5000MS) AND "TON".TON[69].Q;
   END_TRANSITION
   TRANSITION Trans695 FROM RobotTaskSelect TO Grip2SensorError   // T695
      := ((("AutoProcessData".F_Robot3Grip2.PartStatus <> 0) AND "iF-ROOBT3Gripper2Detection-") OR (("AutoProcessData".F_Robot3Grip2.PartStatus = 0) AND "iF-ROOBT3Gripper2Detection-")) AND (#RobotTaskSelect.T > t#5000MS) AND "TON".TON[70].Q;
   END_TRANSITION
   TRANSITION Trans642 FROM RobotTaskSelect TO PressPick   // T637
      := NOT "ChangeOver_DB".Robot_3.MaintenancePosReqSelFlag AND ("AutoProcessData".F_Robot3Grip1.PartStatus = 0) AND NOT "iF-ROOBT3Gripper1Detection" AND "KukaRobot2_CtrlDB".sROBtoPLC.User.Home.DO181_Robot3Area AND NOT "AutoProcessControl".Robot_2.GlueNGPutFlag AND NOT "AutoProcessControl".Robot_2.ScanNGPutFlag AND NOT "AutoProcessControl".Robot_2.Press2PutFlag AND NOT "PalletNGData".UnLoadingNGPallet.OpenFlag AND "AutoProcessControl".B_Press_2.Robot3PickPrimit AND NOT "Robot_DB".Robot_3.MasteringTest_Req AND NOT "Robot_DB".Robot_3.BrakeTest_Req;
   END_TRANSITION
   TRANSITION Trans640 FROM RobotTaskSelect TO PressRingPut   // T634
      := NOT "ChangeOver_DB".Robot_3.MaintenancePosReqSelFlag AND ("AutoProcessData".F_Robot3Grip2.PartStatus = 199) AND NOT "ChangeOver_DB".Global.ManualModeFlag AND ("iF-ROOBT3Gripper2Detection-" OR "AlwaysTRUE") AND NOT "ST10Cylinder".Cy[18].In.HomePositionSensor AND ("AutoProcessData".F_Robot3Grip1.PartStatus = 0) AND NOT "iF-ROOBT3Gripper1Detection" AND NOT "KukaRobot2_CtrlDB".sROBtoPLC.User.Cycle.DO253_GlueNGPutInside AND NOT "KukaRobot2_CtrlDB".sROBtoPLC.User.Cycle.DO249_ScanNGPutInside AND NOT "KukaRobot2_CtrlDB".sROBtoPLC.User.Cycle.DO273_PressPutPart1Inside AND "KukaRobot2_CtrlDB".sROBtoPLC.User.Home.DO181_Robot3Area AND "KukaRobot2_CtrlDB".sROBtoPLC.User.Home.DO180_PressPutArea AND NOT "AutoProcessControl".Robot_2.GlueNGPutFlag AND NOT "AutoProcessControl".Robot_2.ScanNGPutFlag AND NOT "AutoProcessControl".Robot_2.Press2PutFlag AND NOT "PalletNGData".UnLoadingNGPallet.OpenFlag AND "AutoProcessControl".B_Press_2.Robot3PutRingPrimit AND NOT "Robot_DB".Robot_3.MasteringTest_Req AND NOT "Robot_DB".Robot_3.BrakeTest_Req;
   END_TRANSITION
   TRANSITION Trans672 FROM RobotTaskSelect TO OKPut   // T672
      := NOT "ChangeOver_DB".Robot_3.MaintenancePosReqSelFlag AND ("AutoProcessData".F_Robot3Grip1.PartStatus = 499) AND NOT "ChangeOver_DB".Global.ManualModeFlag AND ("iF-ROOBT3Gripper1Detection" OR "AlwaysTRUE") AND NOT "ST10Cylinder".Cy[17].In.HomePositionSensor AND NOT "ST10Cylinder".Cy[17].In.WorkPositionSensor AND NOT "PalletNGData".UnLoadingNGPallet.OpenFlag AND "AutoProcessControl".L_ShafeLine.Robot3PutPrimit;
   END_TRANSITION
   TRANSITION NoUsed FROM RobotTaskSelect TO PressShaftPut   // T631
      := NOT "ChangeOver_DB".Robot_3.MaintenancePosReqSelFlag AND "AlwaysTRUE" AND NOT "AlwaysTRUE" AND ("AutoProcessData".F_Robot3Grip1.PartStatus = 199) AND ("iF-ROOBT3Gripper1Detection" OR "AlwaysTRUE") AND NOT "ST10Cylinder".Cy[17].In.HomePositionSensor AND ("AutoProcessData".F_Robot3Grip2.PartStatus = 199) AND ("iF-ROOBT3Gripper2Detection-" OR "AlwaysTRUE") AND NOT "ST10Cylinder".Cy[18].In.HomePositionSensor AND NOT "PalletNGData".UnLoadingNGPallet.OpenFlag AND "AutoProcessControl".B_Press_1.Robot1PutShaftPrimit;
   END_TRANSITION
   TRANSITION Trans711 FROM RobotTaskSelect TO Maintenance   // T673
      := ((("AutoProcessData".F_Robot3Grip1.PartStatus = 0) AND NOT "iF-ROOBT3Gripper1Detection" AND ("AutoProcessData".F_Robot3Grip2.PartStatus = 0) AND NOT "iF-ROOBT3Gripper2Detection-" AND "ChangeOver_DB".Robot_3.Req_RobotToMaintenancePos) OR ("ChangeOver_DB".Robot_3.HMI_MaintenancePosActive AND NOT "AutoProcessControl".Robot_3.MaintenanceRequest)) AND NOT "Robot_DB".Robot_3.MasteringTest_Req AND NOT "Robot_DB".Robot_3.BrakeTest_Req;
   END_TRANSITION
   TRANSITION Trans902 FROM RobotTaskSelect TO Masref_test   // T902
      := ("AutoProcessData".F_Robot3Grip1.PartStatus = 0) AND NOT "iF-ROOBT3Gripper1Detection" AND "Robot_DB".Robot_3.MasteringTest_Req;
   END_TRANSITION
   TRANSITION Trans903 FROM RobotTaskSelect TO Brake_Test   // T903
      := ("AutoProcessData".F_Robot3Grip1.PartStatus = 0) AND NOT "iF-ROOBT3Gripper1Detection" AND "Robot_DB".Robot_3.BrakeTest_Req;
   END_TRANSITION
   STEP PickPallet:   // S115, max time T#10S, warning time T#7S
              R    #ioPM_Inface.ProcessComplete
              S    #ioPM_Inface.ProcessStart
   END_STEP
   TRANSITION Trans627 FROM PickPallet TO PickPalletProcess   // T115, jump
      := TRUE;
   END_TRANSITION
   STEP PickGlueNGReq:   // S120, max time T#10S, warning time T#7S
              R    #ioPM_Inface.ProcessComplete
              S    #ioPM_Inface.ProcessStart
   END_STEP
   TRANSITION Trans629 FROM PickGlueNGReq TO PickGlueNGProcess   // T120, jump
      := TRUE;
   END_TRANSITION
   STEP PickTable:   // S130, max time T#10S, warning time T#7S
              R    #ioPM_Inface.ProcessComplete
              S    #ioPM_Inface.ProcessStart
   END_STEP
   TRANSITION Trans631 FROM PickTable TO PickTableProcess   // T130, jump
      := TRUE;
   END_TRANSITION
   STEP ScanRing:   // S135, max time T#10S, warning time T#7S
              R    #ioPM_Inface.ProcessComplete
              S    #ioPM_Inface.ProcessStart
   END_STEP
   TRANSITION Trans634 FROM ScanRing TO ScanRingProcess   // T135, jump
      := TRUE;
   END_TRANSITION
   STEP PickMagnetNGReqPick:   // S125, max time T#10S, warning time T#7S
              R    #ioPM_Inface.ProcessComplete
              S    #ioPM_Inface.ProcessStart
   END_STEP
   TRANSITION Trans636 FROM PickMagnetNGReqPick TO MagnScanNGProcess   // T125, jump
      := TRUE;
   END_TRANSITION
   STEP OKPut:   // S155, max time T#10S, warning time T#7S
              R    #ioPM_Inface.ProcessComplete
              S    #ioPM_Inface.ProcessStart
   END_STEP
   TRANSITION Trans649 FROM OKPut TO GluePutProcess   // T155, jump
      := TRUE;
   END_TRANSITION
   STEP PressRingPut:   // S145, max time T#10S, warning time T#7S
              R    #ioPM_Inface.ProcessComplete
              S    #ioPM_Inface.ProcessStart
   END_STEP
   TRANSITION Trans639 FROM PressRingPut TO PressRingPutProcess   // T145, jump
      := TRUE;
   END_TRANSITION
   STEP "NG2Put_1Press/Glue":   // S160, max time T#10S, warning time T#7S
              R    #ioPM_Inface.ProcessComplete
              S    #ioPM_Inface.ProcessStart
   END_STEP
   TRANSITION Trans676 FROM "NG2Put_1Press/Glue" TO "NG PutProcess"   // T160, jump
      := TRUE;
   END_TRANSITION
   STEP "NG2Put_2/Magnet":   // S165, max time T#10S, warning time T#7S
              R    #ioPM_Inface.ProcessComplete
              S    #ioPM_Inface.ProcessStart
   END_STEP
   TRANSITION Trans677 FROM "NG2Put_2/Magnet" TO "NG 2 PutProcess"   // T165, jump
      := TRUE;
   END_TRANSITION
   STEP "NG2Put_3/Ring":   // S170, max time T#10S, warning time T#7S
              R    #ioPM_Inface.ProcessComplete
              S    #ioPM_Inface.ProcessStart
   END_STEP
   TRANSITION Trans679 FROM "NG2Put_3/Ring" TO "NG 3 PutProcess"   // T170, jump
      := TRUE;
   END_TRANSITION
   STEP Grip1SensorError:   // S381, max time T#10S, warning time T#7S
          S1  S    "ST10_DeviceError".F.Robot_3.Grip1SensorCheckError
   END_STEP
   TRANSITION Trans696 FROM Grip1SensorError TO RobotTaskSelect   // T696, jump
      := #iSysInface.Reset;
   END_TRANSITION
   STEP Grip2SensorError:   // S382, max time T#10S, warning time T#7S
          S1  S    "ST10_DeviceError".F.Robot_3.Grip2SensorCheckError
   END_STEP
   TRANSITION Trans697 FROM Grip2SensorError TO RobotTaskSelect   // T697, jump
      := #iSysInface.Reset;
   END_TRANSITION
   STEP PressPick:   // S150, max time T#10S, warning time T#7S
              R    #ioPM_Inface.ProcessComplete
              S    #ioPM_Inface.ProcessStart
   END_STEP
   TRANSITION Trans641 FROM PressPick TO PressPickProcess   // T150, jump
      := TRUE;
   END_TRANSITION
   STEP FlagReset:   // S272, max time T#10S, warning time T#7S
              R    "AutoProcessControl".Robot_3.Press2PutFlag
              R    "AutoProcessControl".Robot_3.Press2PickFlag
              R    "AutoProcessControl".Robot_3.GlueNGPickFlag
              R    "AutoProcessControl".Robot_3.ScanNGPickFlag
              R    "AutoProcessControl".Robot_3.NGPutFlag
   END_STEP
   TRANSITION Trans273 FROM FlagReset TO RobotTaskSelect   // T273
      := NOT "AutoProcessControl".Robot_3.Press2PutFlag AND NOT "AutoProcessControl".Robot_3.Press2PickFlag AND NOT "AutoProcessControl".Robot_3.GlueNGPickFlag AND NOT "AutoProcessControl".Robot_3.ScanNGPickFlag AND NOT "AutoProcessControl".Robot_3.NGPutFlag;
   END_TRANSITION
   STEP Maintenance:   // S131, max time T#10S, warning time T#7S
              R    #ioPM_Inface.ProcessComplete
              S    #ioPM_Inface.ProcessStart
   END_STEP
   TRANSITION Trans710 FROM Maintenance TO "Maintenance Pos"   // T131, jump
      := TRUE;
   END_TRANSITION
   STEP Masref_test:   // S132, max time T#10S, warning time T#7S
              R    #ioPM_Inface.ProcessComplete
              S    #ioPM_Inface.ProcessStart
   END_STEP
   TRANSITION Trans713 FROM Masref_test TO MasteringTest_Req   // T132, jump
      := TRUE;
   END_TRANSITION
   STEP Brake_Test:   // S133, max time T#10S, warning time T#7S
              R    #ioPM_Inface.ProcessComplete
              S    #ioPM_Inface.ProcessStart
   END_STEP
   TRANSITION Trans714 FROM Brake_Test TO BrakeTest_Req   // T133, jump
      := TRUE;
   END_TRANSITION

   // sequencer 3: S200-S249 Fixturecode reading
   STEP "Tablecode Scan":   // S200, max time T#10S, warning time T#7S
   END_STEP
   TRANSITION Trans147 FROM "Tablecode Scan" TO StartRobotScanGripperCode   // T200
      := TRUE;
   END_TRANSITION
   STEP WaitPos4ScanFinish:   // S319, max time T#10S, warning time T#7S
   END_STEP
   TRANSITION Trans628 FROM WaitPos4ScanFinish TO WaitRobotReachPos5   // T641
      := "KukaRobot3_CtrlDB".sPLCtoROB.User.Cycle.DI229_ScanPos4Complete;
   END_TRANSITION
   STEP WaitRobotReachPos3:   // S314, max time T#10S, warning time T#7S
   END_STEP
   TRANSITION P3 FROM WaitRobotReachPos3 TO WaitPos3ScanFinish   // T639
      := "KukaRobot3_CtrlDB".sROBtoPLC.User.Cycle.DO228_ScanPos3Reach;
   END_TRANSITION
   STEP WaitPos6ScanFinish:   // S323, max time T#10S, warning time T#7S
   END_STEP
   TRANSITION Trans644 FROM WaitPos6ScanFinish TO WaitRobotReachPos7   // T644
      := "KukaRobot3_CtrlDB".sPLCtoROB.User.Cycle.DI231_ScanPos6Complete;
   END_TRANSITION
   STEP WaitRobotReachPos5:   // S321, max time T#10S, warning time T#7S
   END_STEP
   TRANSITION P5 FROM WaitRobotReachPos5 TO WaitPos5ScanFinish   // T642
      := "KukaRobot3_CtrlDB".sROBtoPLC.User.Cycle.DO230_ScanPos5Reach;
   END_TRANSITION
   STEP WaitPos5ScanFinish:   // S320, max time T#10S, warning time T#7S
   END_STEP
   TRANSITION Trans643 FROM WaitPos5ScanFinish TO Step380   // T643
      := "KukaRobot3_CtrlDB".sPLCtoROB.User.Cycle.DI230_ScanPos5Complete;
   END_TRANSITION
   STEP WaitPos3ScanFinish:   // S315, max time T#10S, warning time T#7S
   END_STEP
   TRANSITION Trans624 FROM WaitPos3ScanFinish TO WaitRobotReachPos4   // T636
      := "KukaRobot3_CtrlDB".sPLCtoROB.User.Cycle.DI228_ScanPos3Complete;
   END_TRANSITION
   STEP WaitRobotReachPos2:   // S313, max time T#10S, warning time T#7S
   END_STEP
   TRANSITION P2 FROM WaitRobotReachPos2 TO WaitPos2ScanFinish   // T633
      := "KukaRobot3_CtrlDB".sROBtoPLC.User.Cycle.DO227_ScanPos2Reach;
   END_TRANSITION
   STEP StartRobotScanFixtureCode:   // S308, max time T#10S, warning time T#7S
              N    "KukaRobot3_CtrlDB".sPLCtoROB.User.Cycle.DI225_ScanPosReq
   END_STEP
   TRANSITION Trans605 FROM StartRobotScanFixtureCode TO WaitRobotReachPos1   // T605
      := "KukaRobot3_CtrlDB".sROBtoPLC.User.Cycle.DO225_ScanPosInside AND NOT "KukaRobot3_CtrlDB".sROBtoPLC.User.Cycle.DO233_ScanPoseFinish;
   END_TRANSITION
   STEP WaitRobotReachPos4:   // S318, max time T#10S, warning time T#7S
   END_STEP
   TRANSITION P4 FROM WaitRobotReachPos4 TO WaitPos4ScanFinish   // T640
      := "KukaRobot3_CtrlDB".sROBtoPLC.User.Cycle.DO229_ScanPos4Reach;
   END_TRANSITION
   STEP WaitPos1ScanFinish:   // S310, max time T#10S, warning time T#7S
   END_STEP
   TRANSITION Trans622 FROM WaitPos1ScanFinish TO WaitRobotReachPos2   // T621
      := "KukaRobot3_CtrlDB".sPLCtoROB.User.Cycle.DI226_ScanPos1Complete;
   END_TRANSITION
   STEP WaitRobotReachPos1:   // S309, max time T#10S, warning time T#7S
   END_STEP
   TRANSITION P1 FROM WaitRobotReachPos1 TO WaitPos1ScanFinish   // T617
      := "KukaRobot3_CtrlDB".sROBtoPLC.User.Cycle.DO226_ScanPos1Reach;
   END_TRANSITION
   STEP WaitPos2ScanFinish:   // S312, max time T#10S, warning time T#7S
   END_STEP
   TRANSITION Trans623 FROM WaitPos2ScanFinish TO WaitRobotReachPos3   // T624
      := "KukaRobot3_CtrlDB".sPLCtoROB.User.Cycle.DI227_ScanPos2Complete;
   END_TRANSITION
   STEP WaitRobotReachPos6:   // S322, max time T#10S, warning time T#7S
   END_STEP
   TRANSITION P6 FROM WaitRobotReachPos6 TO WaitPos6ScanFinish   // T645
      := "KukaRobot3_CtrlDB".sROBtoPLC.User.Cycle.DO231_ScanPos6Reach;
   END_TRANSITION
   STEP WaitPos7ScanFinish:   // S324, max time T#10S, warning time T#7S
   END_STEP
   TRANSITION Trans645 FROM WaitPos7ScanFinish TO "Wait ScanFinish"   // T646
      := "KukaRobot3_CtrlDB".sPLCtoROB.User.Cycle.DI232_ScanPos7Complete;
   END_TRANSITION
   STEP "Wait ScanFinish":   // S242, max time T#10S, warning time T#7S
   END_STEP
   TRANSITION Trans242 FROM "Wait ScanFinish" TO "Tablecode ScanFinish"   // T242
      := "KukaRobot3_CtrlDB".sROBtoPLC.User.Cycle.DO233_ScanPoseFinish;
   END_TRANSITION
   STEP WaitRobotReachPos7:   // S325, max time T#10S, warning time T#7S
   END_STEP
   TRANSITION P7 FROM WaitRobotReachPos7 TO WaitPos7ScanFinish   // T647
      := "KukaRobot3_CtrlDB".sROBtoPLC.User.Cycle.DO232_ScanPos7Reach;
   END_TRANSITION
   STEP "Tablecode ScanFinish":   // S149, max time T#10S, warning time T#7S
              S    #ioPM_Inface.ProcessComplete
              R    #ioPM_Inface.ProcessStart
   END_STEP
   TRANSITION Trans352 FROM "Tablecode ScanFinish" TO ProcessStart   // T149, jump
      := "ChangeOver_DB".Global.AllFixtureScanCompareOk OR "ChangeOver_DB".Robot_3.Req_RobotToMaintenancePos;
   END_TRANSITION
   STEP Step380:   // S380, max time T#10S, warning time T#7S
   END_STEP
   TRANSITION Trans692 FROM Step380 TO WaitRobotReachPos6   // T692
      := "AlwaysTRUE" AND NOT "AlwaysTRUE";
   END_TRANSITION
   TRANSITION Trans693 FROM Step380 TO "Tablecode ScanFinish"   // T693
      := "AlwaysTRUE";
   END_TRANSITION
   STEP StartRobotScanGripperCode:   // S334, max time T#10S, warning time T#7S
              N    "KukaRobot3_CtrlDB".sPLCtoROB.User.Cycle.DI305_GripScan
   END_STEP
   TRANSITION Trans684 FROM StartRobotScanGripperCode TO RobotScanGripperReachPos1   // T616
      := "KukaRobot3_CtrlDB".sROBtoPLC.User.Cycle.DO305_GripScanInside AND NOT "KukaRobot3_CtrlDB".sROBtoPLC.User.Cycle.DO306_GripScanFinish;
   END_TRANSITION
   STEP RobotScanGripperReachPos1:   // S335, max time T#10S, warning time T#7S
   END_STEP
   TRANSITION Trans685 FROM RobotScanGripperReachPos1 TO WaitGripperPos1ScanFinish   // T619
      := "KukaRobot3_CtrlDB".sROBtoPLC.User.Cycle.DO307_ScanPos1Reach;
   END_TRANSITION
   STEP WaitGripperPos1ScanFinish:   // S336, max time T#10S, warning time T#7S
   END_STEP
   TRANSITION Trans686 FROM WaitGripperPos1ScanFinish TO RobotScanGripperReachPos2   // T622
      := "KukaRobot3_CtrlDB".sPLCtoROB.User.Cycle.DI306_ScanPartComplete;
   END_TRANSITION
   STEP RobotScanGripperReachPos2:   // S337, max time T#10S, warning time T#7S
   END_STEP
   TRANSITION Trans687 FROM RobotScanGripperReachPos2 TO WaitGripperPos2ScanFinish   // T623
      := "KukaRobot3_CtrlDB".sROBtoPLC.User.Cycle.DO308_ScanPos2Reach;
   END_TRANSITION
   STEP WaitGripperPos2ScanFinish:   // S338, max time T#10S, warning time T#7S
   END_STEP
   TRANSITION Trans688 FROM WaitGripperPos2ScanFinish TO RobotScanGripperReachPos3   // T626
      := "KukaRobot3_CtrlDB".sPLCtoROB.User.Cycle.DI306_ScanPartComplete;
   END_TRANSITION
   STEP RobotScanGripperReachPos3:   // S339, max time T#10S, warning time T#7S
   END_STEP
   TRANSITION Trans689 FROM RobotScanGripperReachPos3 TO WaitGripperPos3ScanFinish   // T628
      := "KukaRobot3_CtrlDB".sROBtoPLC.User.Cycle.DO309_ScanPos3Reach;
   END_TRANSITION
   STEP WaitGripperPos3ScanFinish:   // S340, max time T#10S, warning time T#7S
   END_STEP
   TRANSITION Trans690 FROM WaitGripperPos3ScanFinish TO RobotScanGripperReachPos4   // T630
      := "KukaRobot3_CtrlDB".sPLCtoROB.User.Cycle.DI306_ScanPartComplete;
   END_TRANSITION
   STEP RobotScanGripperReachPos4:   // S341, max time T#10S, warning time T#7S
   END_STEP
   TRANSITION Trans703 FROM RobotScanGripperReachPos4 TO WaitGripperPos4ScanFinish   // T632
      := "KukaRobot3_CtrlDB".sROBtoPLC.User.Cycle.DO310_ScanPos4Reach;
   END_TRANSITION
   STEP WaitGripperPos4ScanFinish:   // S342, max time T#10S, warning time T#7S
   END_STEP
   TRANSITION Trans704 FROM WaitGripperPos4ScanFinish TO StartRobotScanFixtureCode   // T635
      := "KukaRobot3_CtrlDB".sROBtoPLC.User.Cycle.DO306_GripScanFinish AND "AutoProcessControl".Fixture2Code.Robot3CodeReadReq;
   END_TRANSITION

   // sequencer 4: S250-S299 PickPallet
   STEP PickPalletProcess:   // S250, max time T#10S, warning time T#7S
   END_STEP
   TRANSITION Trans150 FROM PickPalletProcess TO DataClear   // T250
      := TRUE;
   END_TRANSITION
   STEP StartRobotPickPalletShaft:   // S326, max time T#10S, warning time T#7S
              N    "KukaRobot3_CtrlDB".sPLCtoROB.User.Cycle.DI241_PickPalletReq
   END_STEP
   TRANSITION Trans607 FROM StartRobotPickPalletShaft TO WaitRobotGripHaveStatus   // T648
      := "KukaRobot3_CtrlDB".sROBtoPLC.User.Cycle.DO241_PickPalletInside AND NOT "KukaRobot3_CtrlDB".sROBtoPLC.User.Cycle.DO242_PickPalletFinish;
   END_TRANSITION
   STEP WaitRobotFinish:   // S327, max time T#10S, warning time T#7S
   END_STEP
   TRANSITION P8 FROM WaitRobotFinish TO PickPalletFinish   // T327
      := "KukaRobot3_CtrlDB".sROBtoPLC.User.Cycle.DO242_PickPalletFinish;
   END_TRANSITION
   STEP PickPalletFinish:   // S299, max time T#10S, warning time T#7S
              S    #ioPM_Inface.ProcessComplete
              R    #ioPM_Inface.ProcessStart
   END_STEP
   TRANSITION Trans654 FROM PickPalletFinish TO ProcessStart   // T299, jump
      := TRUE;
   END_TRANSITION
   STEP WaitRobotGripHaveStatus:   // S346, max time T#10S, warning time T#7S
   END_STEP
   TRANSITION Trans655 FROM WaitRobotGripHaveStatus TO Grip1PartStatus   // T655
      := "KukaRobot3_CtrlDB".sROBtoPLC.User.Public.GO5_RobGrip1Status <> 0;
   END_TRANSITION
   STEP Grip1PartStatus:   // S243, max time T#10S, warning time T#7S
              N    "AutoProcessData".F_Robot3Grip1.PartStatus:=100
   END_STEP
   TRANSITION Trans243 FROM Grip1PartStatus TO WaitRobotFinish   // T243
      := "AutoProcessData".F_Robot3Grip1.PartStatus = 100;
   END_TRANSITION
   STEP DataClear:   // S252, max time T#10S, warning time T#7S
          S1  N    "AutoProcessData".F_Robot3Grip1:="AutoProcessData".ClearData
   END_STEP
   TRANSITION Trans253 FROM DataClear TO StartRobotPickPalletShaft   // T253
      := TRUE;
   END_TRANSITION

   // sequencer 5: S300-S349 PickGlueNGR
   STEP PickGlueNGProcess:   // S300, max time T#10S, warning time T#7S
   END_STEP
   TRANSITION Trans300 FROM PickGlueNGProcess TO StartRobotPickGlueNG   // T300
      := TRUE;
   END_TRANSITION
   STEP DataMove:   // S253, max time T#10S, warning time T#7S
          S1  N    "AutoProcessData".F_Robot3Grip1:="AutoProcessData".C_GlueNGBuffer
          S1  N    "AutoProcessData".C_GlueNGBuffer:="AutoProcessData".ClearData
   END_STEP
   TRANSITION Trans254 FROM DataMove TO WaitRobotFinish_1   // T254
      := #DataMove.T > t#100MS;
   END_TRANSITION
   STEP StartRobotPickGlueNG:   // S328, max time T#10S, warning time T#7S
              N    "KukaRobot3_CtrlDB".sPLCtoROB.User.Cycle.DI253_PickGlueNGReq
   END_STEP
   TRANSITION Trans610 FROM StartRobotPickGlueNG TO WaitRobotGripHaveStatus_1   // T328
      := "KukaRobot3_CtrlDB".sROBtoPLC.User.Cycle.DO253_PickGlueNGInside AND NOT "KukaRobot3_CtrlDB".sROBtoPLC.User.Cycle.DO254_PickGlueNGFinish;
   END_TRANSITION
   STEP WaitRobotFinish_1:   // S343, max time T#10S, warning time T#7S
   END_STEP
   TRANSITION P9 FROM WaitRobotFinish_1 TO PickGlueNGFinish_1   // T651
      := "KukaRobot3_CtrlDB".sROBtoPLC.User.Cycle.DO254_PickGlueNGFinish;
   END_TRANSITION
   STEP PickGlueNGFinish_1:   // S349, max time T#10S, warning time T#7S
              S    #ioPM_Inface.ProcessComplete
              R    #ioPM_Inface.ProcessStart
   END_STEP
   TRANSITION Trans656 FROM PickGlueNGFinish_1 TO ProcessStart   // T349, jump
      := TRUE;
   END_TRANSITION
   STEP WaitRobotGripHaveStatus_1:   // S347, max time T#10S, warning time T#7S
   END_STEP
   TRANSITION Trans657 FROM WaitRobotGripHaveStatus_1 TO DataMove   // T656
      := "KukaRobot3_CtrlDB".sROBtoPLC.User.Public.GO5_RobGrip1Status <> 0;
   END_TRANSITION

   // sequencer 6: S350-S399 MagnScanNG
   STEP MagnScanNGProcess:   // S350, max time T#10S, warning time T#7S
   END_STEP
   TRANSITION Trans350 FROM MagnScanNGProcess TO StartRobotPickMagnScanNG   // T350
      := TRUE;
   END_TRANSITION
   STEP DataMove_1:   // S255, max time T#10S, warning time T#7S
          S1  N    "AutoProcessData".F_Robot3Grip2:="AutoProcessData".C_MagnScanNGBuffer
          S1  N    "AutoProcessData".C_MagnScanNGBuffer:="AutoProcessData".ClearData
   END_STEP
   TRANSITION Trans256 FROM DataMove_1 TO WaitRobotFinish_2   // T256
      := #DataMove_1.T > t#100MS;
   END_TRANSITION
   STEP StartRobotPickMagnScanNG:   // S344, max time T#10S, warning time T#7S
              N    "KukaRobot3_CtrlDB".sPLCtoROB.User.Cycle.DI249_PickMagnetNGReq
   END_STEP
   TRANSITION Trans611 FROM StartRobotPickMagnScanNG TO WaitRobotGripHaveStatus_2   // T652
      := "KukaRobot3_CtrlDB".sROBtoPLC.User.Cycle.DO249_PickMagnetInside AND NOT "KukaRobot3_CtrlDB".sROBtoPLC.User.Cycle.DO250_PickMagnetFinish;
   END_TRANSITION
   STEP WaitRobotFinish_2:   // S345, max time T#10S, warning time T#7S
   END_STEP
   TRANSITION P10 FROM WaitRobotFinish_2 TO Step930   // T653
      := "KukaRobot3_CtrlDB".sROBtoPLC.User.Cycle.DO250_PickMagnetFinish;
   END_TRANSITION
   STEP PickMagnScanNGBufferFinish:   // S399, max time T#10S, warning time T#7S
              S    #ioPM_Inface.ProcessComplete
              R    #ioPM_Inface.ProcessStart
   END_STEP
   TRANSITION Trans658 FROM PickMagnScanNGBufferFinish TO ProcessStart   // T399, jump
      := TRUE;
   END_TRANSITION
   STEP WaitRobotGripHaveStatus_2:   // S348, max time T#10S, warning time T#7S
   END_STEP
   TRANSITION Trans659 FROM WaitRobotGripHaveStatus_2 TO DataMove_1   // T657
      := "KukaRobot3_CtrlDB".sROBtoPLC.User.Public.GO6_RobGrip2Status <> 0;
   END_TRANSITION
   STEP Step930:   // S930, max time T#10S, warning time T#7S
              N    "AutoProcessData".F_Robot3Grip1.PartStatus:=444
   END_STEP
   TRANSITION Trans930 FROM Step930 TO PickMagnScanNGBufferFinish   // T930
      := #Step930.T > t#100MS;
   END_TRANSITION

   // sequencer 7: S400-S449 PickTable
   STEP PickTableProcess:   // S400, max time T#10S, warning time T#7S
   END_STEP
   TRANSITION Trans400 FROM PickTableProcess TO "Data Clear_2"   // T400
      := TRUE;
   END_TRANSITION
   STEP Grip2PartStatus:   // S244, max time T#10S, warning time T#7S
              N    "AutoProcessData".F_Robot3Grip2.PartStatus:=100
   END_STEP
   TRANSITION Trans244 FROM Grip2PartStatus TO WaitRobotFinish_3   // T244
      := "AutoProcessData".F_Robot3Grip2.PartStatus = 100;
   END_TRANSITION
   STEP StartRobotPickTable:   // S352, max time T#10S, warning time T#7S
              N    "KukaRobot3_CtrlDB".sPLCtoROB.User.Cycle.DI257_PickTableReq
   END_STEP
   TRANSITION Trans618 FROM StartRobotPickTable TO WaitRobotGripHaveStatus_3   // T654
      := "KukaRobot3_CtrlDB".sROBtoPLC.User.Cycle.DO257_PickTableInside AND NOT "KukaRobot3_CtrlDB".sROBtoPLC.User.Cycle.DO258_PickTableFinish;
   END_TRANSITION
   STEP WaitRobotFinish_3:   // S353, max time T#10S, warning time T#7S
   END_STEP
   TRANSITION P11 FROM WaitRobotFinish_3 TO PickTableProcessFinish   // T658
      := "KukaRobot3_CtrlDB".sROBtoPLC.User.Cycle.DO258_PickTableFinish;
   END_TRANSITION
   STEP PickTableProcessFinish:   // S449, max time T#10S, warning time T#7S
              S    #ioPM_Inface.ProcessComplete
              R    #ioPM_Inface.ProcessStart
   END_STEP
   TRANSITION Trans660 FROM PickTableProcessFinish TO ProcessStart   // T449, jump
      := TRUE;
   END_TRANSITION
   STEP WaitRobotGripHaveStatus_3:   // S354, max time T#10S, warning time T#7S
   END_STEP
   TRANSITION Trans661 FROM WaitRobotGripHaveStatus_3 TO Grip2PartStatus   // T659
      := "KukaRobot3_CtrlDB".sROBtoPLC.User.Public.GO6_RobGrip2Status <> 0;
   END_TRANSITION
   STEP "Data Clear_2":   // S258, max time T#10S, warning time T#7S
          S1  N    "AutoProcessData".F_Robot3Grip2:="AutoProcessData".ClearData
   END_STEP
   TRANSITION Trans259 FROM "Data Clear_2" TO StartRobotPickTable   // T259
      := #"Data Clear_2".T > t#100MS;
   END_TRANSITION

   // sequencer 8: S450-S499 ScanRing
   STEP ScanRingProcess:   // S450, max time T#10S, warning time T#7S
   END_STEP
   TRANSITION Trans450 FROM ScanRingProcess TO StartRobotScanRing   // T450
      := TRUE;
   END_TRANSITION
   STEP CheckScanReady:   // S245, max time T#10S, warning time T#7S
   END_STEP
   TRANSITION Trans245 FROM CheckScanReady TO ScanStart   // T245
      := "KeyenceSR1000Ctrl_803A1DB".oReady;
   END_TRANSITION
   STEP StartRobotScanRing:   // S355, max time T#10S, warning time T#7S
              N    "KukaRobot3_CtrlDB".sPLCtoROB.User.Cycle.DI261_ScanRingReq
   END_STEP
   TRANSITION Trans619 FROM StartRobotScanRing TO WaitRobotReachScanPos   // T660
      := "KukaRobot3_CtrlDB".sROBtoPLC.User.Cycle.DO261_ScanRingtInside AND NOT "KukaRobot3_CtrlDB".sROBtoPLC.User.Cycle.DO262_ScanRingFinish;
   END_TRANSITION
   STEP WaitRobotFinish_4:   // S356, max time T#10S, warning time T#7S
              N    "KukaRobot3_CtrlDB".sPLCtoROB.User.Cycle.DI262_ScanRingComplete
   END_STEP
   TRANSITION P12 FROM WaitRobotFinish_4 TO ScanRingProcessFinish   // T661
      := "KukaRobot3_CtrlDB".sROBtoPLC.User.Cycle.DO262_ScanRingFinish;
   END_TRANSITION
   STEP ScanRingProcessFinish:   // S499, max time T#10S, warning time T#7S
              S    #ioPM_Inface.ProcessComplete
              R    #ioPM_Inface.ProcessStart
   END_STEP
   TRANSITION Trans662 FROM ScanRingProcessFinish TO ProcessStart   // T499, jump
      := TRUE;
   END_TRANSITION
   STEP WaitRobotReachScanPos:   // S357, max time T#10S, warning time T#7S
   END_STEP
   TRANSITION Trans663 FROM WaitRobotReachScanPos TO CheckScanReady   // T662
      := "KukaRobot3_CtrlDB".sROBtoPLC.User.Cycle.DO263_ScanReach;
   END_TRANSITION
   STEP ScanStart:   // S246, max time T#10S, warning time T#7S
          S1  S    "KeyenceSR1000Ctrl_803A1DB".ioAutoTrigger
   END_STEP
   TRANSITION Trans246 FROM ScanStart TO WaitScanCompletely   // T246
      := NOT "KeyenceSR1000Ctrl_803A1DB".sHMI.Status.Ready;
   END_TRANSITION
   STEP WaitScanCompletely:   // S247, max time T#10S, warning time T#7S
   END_STEP
   TRANSITION Trans247 FROM WaitScanCompletely TO CodeMove   // T247
      := "KeyenceSR1000Ctrl_803A1DB".sHMI.Status.Complete AND "KeyenceSR1000Ctrl_803A1DB".sHMI.Status.ReadOk;
   END_TRANSITION
   TRANSITION Trans248 FROM WaitScanCompletely TO PartNGStatus   // T248
      := "KeyenceSR1000Ctrl_803A1DB".sHMI.Status.Complete AND "KeyenceSR1000Ctrl_803A1DB".sHMI.Status.ReadNok;
   END_TRANSITION
   STEP CodeMove:   // S248, max time T#10S, warning time T#7S
              N    "AutoProcessData".F_Robot3Grip2.RingCode_2:="KeyenceSR1000Ctrl_803A1DB".sHMI.Status.CurrentCode
   END_STEP
   TRANSITION Trans249 FROM CodeMove TO PartOKStatus_1   // T249
      := TRUE;
   END_TRANSITION
   STEP PartOKStatus:   // S249, max time T#10S, warning time T#7S
              N    "AutoProcessData".F_Robot3Grip2.PartStatus:=199
   END_STEP
   TRANSITION Trans251 FROM PartOKStatus TO WaitRobotFinish_4   // T251
      := "AutoProcessData".F_Robot3Grip2.PartStatus = 199;
   END_TRANSITION
   STEP PartNGStatus:   // S251, max time T#10S, warning time T#7S
              N    "AutoProcessData".F_Robot3Grip2.PartStatus:=150
   END_STEP
   TRANSITION Trans252 FROM PartNGStatus TO WaitRobotFinish_4   // T252
      := "AutoProcessData".F_Robot3Grip2.PartStatus = 150;
   END_TRANSITION
   STEP "MES Online  offline?":   // S385, max time T#10S, warning time T#7S
   END_STEP
   TRANSITION Offline FROM "MES Online  offline?" TO PartOKStatus   // T702
      := "Station_Sys".Cmd.OnOffLine;
   END_TRANSITION
   TRANSITION Trans702 FROM "MES Online  offline?" TO WaitRobotFinish_4   // T704
      := NOT "Station_Sys".Cmd.OnOffLine;
   END_TRANSITION
   STEP PartOKStatus_1:   // S273, max time T#10S, warning time T#7S
              N    "AutoProcessData".F_Robot3Grip2.PartStatus:=110
   END_STEP
   TRANSITION Trans274 FROM PartOKStatus_1 TO "MES Online  offline?"   // T274
      := "AutoProcessData".F_Robot3Grip2.PartStatus = 110;
   END_TRANSITION

   // sequencer 9: S500-S549 PressShaftPut
   STEP PressShaftPutProcess:   // S500, max time T#10S, warning time T#7S
   END_STEP
   TRANSITION Trans500 FROM PressShaftPutProcess TO StartRobotPressShaftPut   // T500
      := TRUE;
   END_TRANSITION
   STEP DataMove_2:   // S257, max time T#10S, warning time T#7S
          S1  N    "AutoProcessData".B_Press2:="AutoProcessData".F_Robot3Grip1
          S1  N    "AutoProcessData".F_Robot3Grip1:="AutoProcessData".ClearData
   END_STEP
   TRANSITION Trans258 FROM DataMove_2 TO WaitRobotFinish_5   // T258
      := #DataMove_2.T > t#100MS;
   END_TRANSITION
   STEP StartRobotPressShaftPut:   // S358, max time T#10S, warning time T#7S
              N    "KukaRobot3_CtrlDB".sPLCtoROB.User.Cycle.DI273_PressPutPart1Req
   END_STEP
   TRANSITION Trans646 FROM StartRobotPressShaftPut TO WaitRobotGripStatus   // T663
      := "KukaRobot3_CtrlDB".sROBtoPLC.User.Cycle.DO273_PressPutPart1Inside AND NOT "KukaRobot3_CtrlDB".sROBtoPLC.User.Cycle.DO274_PressPutPart1Finish;
   END_TRANSITION
   STEP WaitRobotFinish_5:   // S359, max time T#10S, warning time T#7S
   END_STEP
   TRANSITION P13 FROM WaitRobotFinish_5 TO PressShaftPutProcessFinish   // T664
      := "KukaRobot3_CtrlDB".sROBtoPLC.User.Cycle.DO274_PressPutPart1Finish;
   END_TRANSITION
   STEP PressShaftPutProcessFinish:   // S549, max time T#10S, warning time T#7S
              S    #ioPM_Inface.ProcessComplete
              R    #ioPM_Inface.ProcessStart
   END_STEP
   TRANSITION Trans664 FROM PressShaftPutProcessFinish TO ProcessStart   // T549, jump
      := TRUE;
   END_TRANSITION
   STEP WaitRobotGripStatus:   // S360, max time T#10S, warning time T#7S
   END_STEP
   TRANSITION Trans665 FROM WaitRobotGripStatus TO DataMove_2   // T665
      := "KukaRobot3_CtrlDB".sROBtoPLC.User.Public.GO5_RobGrip1Status = 0;
   END_TRANSITION

   // sequencer 10: S550-S599 PressRingPut
   STEP PressRingPutProcess:   // S550, max time T#10S, warning time T#7S
   END_STEP
   TRANSITION Trans550 FROM PressRingPutProcess TO StartRobotPressRingPut   // T550
      := TRUE;
   END_TRANSITION
   STEP DataMove_3:   // S260, max time T#10S, warning time T#7S
              N    "AutoProcessData".B_Press2.RingCode_2:="AutoProcessData".F_Robot3Grip2.RingCode_2
              N    "AutoProcessData".B_Press2.PartStatus:=420
   END_STEP
   TRANSITION Trans261 FROM DataMove_3 TO "Data Clear_4"   // T261
      := (#DataMove_3.T > t#100MS) AND ("AutoProcessData".B_Press2.PartStatus = 420);
   END_TRANSITION
   STEP StartRobotPressRingPut:   // S361, max time T#10S, warning time T#7S
              N    "KukaRobot3_CtrlDB".sPLCtoROB.User.Cycle.DI277_PressPutRingReq
   END_STEP
   TRANSITION Trans647 FROM StartRobotPressRingPut TO WaitRobotGripStatus_1   // T666
      := "KukaRobot3_CtrlDB".sROBtoPLC.User.Cycle.DO277_PressPutRingInside AND NOT "KukaRobot3_CtrlDB".sROBtoPLC.User.Cycle.DO278_PressPutRingFinish;
   END_TRANSITION
   STEP WaitRobotFinish_6:   // S362, max time T#10S, warning time T#7S
   END_STEP
   TRANSITION P14 FROM WaitRobotFinish_6 TO PressRingPutProcessFinish   // T667
      := "KukaRobot3_CtrlDB".sROBtoPLC.User.Cycle.DO278_PressPutRingFinish;
   END_TRANSITION
   STEP PressRingPutProcessFinish:   // S599, max time T#10S, warning time T#7S
              S    #ioPM_Inface.ProcessComplete
              R    #ioPM_Inface.ProcessStart
   END_STEP
   TRANSITION Trans666 FROM PressRingPutProcessFinish TO ProcessStart   // T599, jump
      := TRUE;
   END_TRANSITION
   STEP WaitRobotGripStatus_1:   // S363, max time T#10S, warning time T#7S
   END_STEP
   TRANSITION Trans667 FROM WaitRobotGripStatus_1 TO DataMove_3   // T668
      := "KukaRobot3_CtrlDB".sROBtoPLC.User.Public.GO6_RobGrip2Status = 0;
   END_TRANSITION
   STEP "Data Clear_4":   // S261, max time T#10S, warning time T#7S
          S1  N    "AutoProcessData".F_Robot3Grip2:="AutoProcessData".ClearData
   END_STEP
   TRANSITION Trans262 FROM "Data Clear_4" TO WaitRobotFinish_6   // T262
      := TRUE;
   END_TRANSITION

   // sequencer 11: S600-S649 PressPick
   STEP PressPickProcess:   // S600, max time T#10S, warning time T#7S
   END_STEP
   TRANSITION Trans600 FROM PressPickProcess TO StartRobotPressPick   // T600
      := TRUE;
   END_TRANSITION
   STEP DataMove_4:   // S262, max time T#10S, warning time T#7S
          S1  N    "AutoProcessData".F_Robot3Grip1:="AutoProcessData".B_Press2
          S1  N    "AutoProcessData".B_Press2:="AutoProcessData".ClearData
   END_STEP
   TRANSITION Trans263 FROM DataMove_4 TO WaitRobotFinish_7   // T263
      := #DataMove_4.T > t#100MS;
   END_TRANSITION
   STEP StartRobotPressPick:   // S364, max time T#10S, warning time T#7S
              N    "KukaRobot3_CtrlDB".sPLCtoROB.User.Cycle.DI281_PressPickPartReq
   END_STEP
   TRANSITION Trans648 FROM StartRobotPressPick TO WaitRobotGripStatus_2   // T669
      := "KukaRobot3_CtrlDB".sROBtoPLC.User.Cycle.DO281_PressPickInside AND NOT "KukaRobot3_CtrlDB".sROBtoPLC.User.Cycle.DO282_PressPickFinish;
   END_TRANSITION
   STEP WaitRobotFinish_7:   // S365, max time T#10S, warning time T#7S
   END_STEP
   TRANSITION P15 FROM WaitRobotFinish_7 TO PressPickProcessFinish_   // T670
      := "KukaRobot3_CtrlDB".sROBtoPLC.User.Cycle.DO282_PressPickFinish;
   END_TRANSITION
   STEP PressPickProcessFinish_:   // S649, max time T#10S, warning time T#7S
              S    #ioPM_Inface.ProcessComplete
              R    #ioPM_Inface.ProcessStart
   END_STEP
   TRANSITION Trans668 FROM PressPickProcessFinish_ TO ProcessStart   // T649, jump
      := TRUE;
   END_TRANSITION
   STEP WaitRobotGripStatus_2:   // S366, max time T#10S, warning time T#7S
   END_STEP
   TRANSITION Trans669 FROM WaitRobotGripStatus_2 TO DataMove_4   // T671
      := "KukaRobot3_CtrlDB".sROBtoPLC.User.Public.GO5_RobGrip1Status <> 0;
   END_TRANSITION

   // sequencer 12: S650-S699 OKPut
   STEP GluePutProcess:   // S650, max time T#10S, warning time T#7S
   END_STEP
   TRANSITION Trans674 FROM GluePutProcess TO StartRobotGluePut   // T650
      := TRUE;
   END_TRANSITION
   STEP DataMove_5:   // S264, max time T#10S, warning time T#7S
          S1  N    "AutoProcessData_Buffer".DataBuffer["AutoProcessData".GlobalData.DataIndex]:="AutoProcessData".F_Robot3Grip1
          S1  N    "AutoProcessData".F_Robot3Grip1:="AutoProcessData".ClearData
          S0  N    "AutoProcessData".GlobalData.DataIndex:="AutoProcessData".GlobalData.DataIndex+1
   END_STEP
   TRANSITION Trans265 FROM DataMove_5 TO "Data Clear_6"   // T265
      := #DataMove_5.T > t#100MS;
   END_TRANSITION
   STEP StartRobotGluePut:   // S367, max time T#10S, warning time T#7S
              N    "KukaRobot3_CtrlDB".sPLCtoROB.User.Cycle.DI289_PutOkPartReq
   END_STEP
   TRANSITION Trans650 FROM StartRobotGluePut TO WaitRobotGripStatus_3   // T676
      := "KukaRobot3_CtrlDB".sROBtoPLC.User.Cycle.DO289_PutOkPartInside AND NOT "KukaRobot3_CtrlDB".sROBtoPLC.User.Cycle.DO290_PutOkPartFinish;
   END_TRANSITION
   STEP WaitRobotFinish_8:   // S368, max time T#10S, warning time T#7S
   END_STEP
   TRANSITION P16 FROM WaitRobotFinish_8 TO OKPutProcessFinish   // T677
      := "KukaRobot3_CtrlDB".sROBtoPLC.User.Cycle.DO290_PutOkPartFinish;
   END_TRANSITION
   STEP OKPutProcessFinish:   // S699, max time T#10S, warning time T#7S
              S    #ioPM_Inface.ProcessComplete
              R    #ioPM_Inface.ProcessStart
   END_STEP
   TRANSITION Trans670 FROM OKPutProcessFinish TO ProcessStart   // T699, jump
      := TRUE;
   END_TRANSITION
   STEP WaitRobotGripStatus_3:   // S369, max time T#10S, warning time T#7S
   END_STEP
   TRANSITION Trans671 FROM WaitRobotGripStatus_3 TO DataMove_5   // T679
      := "KukaRobot3_CtrlDB".sROBtoPLC.User.Public.GO5_RobGrip1Status = 0;
   END_TRANSITION
   STEP "Data Clear_6":   // S265, max time T#10S, warning time T#7S
      // CJ - check
              N    "Robot_DB".Robot_3.SpeedCount:="Robot_DB".Robot_3.SpeedCount+1
   END_STEP
   TRANSITION Trans266 FROM "Data Clear_6" TO WaitRobotFinish_8   // T266
      := TRUE;
   END_TRANSITION

   // sequencer 13: S700-S749 Press/GlueNG1 Put
   STEP "NG PutProcess":   // S700, max time T#10S, warning time T#7S
   END_STEP
   TRANSITION Trans700 FROM "NG PutProcess" TO StartRobotNGPut   // T700
      := TRUE;
   END_TRANSITION
   STEP StartRobotNGPut:   // S370, max time T#10S, warning time T#7S
              N    "KukaRobot3_CtrlDB".sPLCtoROB.User.Cycle.DI265_LoadPressNGReq1
   END_STEP
   TRANSITION Trans651 FROM StartRobotNGPut TO WaitRobotGripStatus_4   // T680
      := "KukaRobot3_CtrlDB".sROBtoPLC.User.Cycle.DO265_LoadNGInside AND NOT "KukaRobot3_CtrlDB".sROBtoPLC.User.Cycle.DO266_LoadNGFinish;
   END_TRANSITION
   STEP WaitRobotFinish_9:   // S371, max time T#10S, warning time T#7S
   END_STEP
   TRANSITION P17 FROM WaitRobotFinish_9 TO "NG1 PutProcessFinish"   // T681
      := "KukaRobot3_CtrlDB".sROBtoPLC.User.Cycle.DO266_LoadNGFinish;
   END_TRANSITION
   STEP "NG1 PutProcessFinish":   // S749, max time T#10S, warning time T#7S
              S    #ioPM_Inface.ProcessComplete
              R    #ioPM_Inface.ProcessStart
   END_STEP
   TRANSITION Trans673 FROM "NG1 PutProcessFinish" TO ProcessStart   // T749, jump
      := TRUE;
   END_TRANSITION
   STEP WaitRobotGripStatus_4:   // S372, max time T#10S, warning time T#7S
   END_STEP
   TRANSITION Trans678 FROM WaitRobotGripStatus_4 TO DataMove_6   // T682
      := "KukaRobot3_CtrlDB".sROBtoPLC.User.Public.GO5_RobGrip1Status = 0;
   END_TRANSITION
   STEP "Data Clear_7":   // S267, max time T#10S, warning time T#7S
          S1  N    "AutoProcessData".F_Robot3Grip1:="AutoProcessData".ClearData
   END_STEP
   TRANSITION Trans268 FROM "Data Clear_7" TO WaitRobotFinish_9   // T268
      := TRUE;
   END_TRANSITION
   STEP DataMove_6:   // S266, max time T#10S, warning time T#7S
                   //"AutoProcessData_Buffer".DataBuffer["AutoProcessData".GlobalData.DataIndex]:="AutoProcessData".F_Robot3Grip1
                   //"AutoProcessData".GlobalData.DataIndex:="AutoProcessData".GlobalData.DataIndex+1
   END_STEP
   TRANSITION Trans267 FROM DataMove_6 TO "Data Clear_7"   // T267
      := #DataMove_6.T > t#100MS;
   END_TRANSITION

   // sequencer 14: S750-S799 Magnet ScanNG2 Put
   STEP "Data Clear_8":   // S268, max time T#10S, warning time T#7S
              N    "AutoProcessData".F_Robot3Grip2:="AutoProcessData".ClearData
   END_STEP
   TRANSITION Trans269 FROM "Data Clear_8" TO WaitRobotFinish_10   // T269
      := TRUE;
   END_TRANSITION
   STEP "NG 2 PutProcess":   // S750, max time T#10S, warning time T#7S
   END_STEP
   TRANSITION Trans701 FROM "NG 2 PutProcess" TO StartRobotNG2Put_1   // T750
      := TRUE;
   END_TRANSITION
   STEP StartRobotNG2Put_1:   // S373, max time T#10S, warning time T#7S
              N    "KukaRobot3_CtrlDB".sPLCtoROB.User.Cycle.DI266_LoadGlueNGReq2
   END_STEP
   TRANSITION Trans652 FROM StartRobotNG2Put_1 TO WaitRobotGripStatus_5   // T685
      := "KukaRobot3_CtrlDB".sROBtoPLC.User.Cycle.DO265_LoadNGInside AND NOT "KukaRobot3_CtrlDB".sROBtoPLC.User.Cycle.DO266_LoadNGFinish;
   END_TRANSITION
   STEP WaitRobotFinish_10:   // S374, max time T#10S, warning time T#7S
   END_STEP
   TRANSITION P18 FROM WaitRobotFinish_10 TO "NG2 PutProcessFinish"   // T686
      := "KukaRobot3_CtrlDB".sROBtoPLC.User.Cycle.DO266_LoadNGFinish;
   END_TRANSITION
   STEP "NG2 PutProcessFinish":   // S799, max time T#10S, warning time T#7S
              S    #ioPM_Inface.ProcessComplete
              R    #ioPM_Inface.ProcessStart
              N    "AutoProcessData".F_Robot3Grip1.PartStatus:=0
   END_STEP
   TRANSITION Trans680 FROM "NG2 PutProcessFinish" TO ProcessStart   // T799, jump
      := TRUE;
   END_TRANSITION
   STEP WaitRobotGripStatus_5:   // S375, max time T#10S, warning time T#7S
   END_STEP
   TRANSITION Trans681 FROM WaitRobotGripStatus_5 TO DataMove_7   // T687
      := "KukaRobot3_CtrlDB".sROBtoPLC.User.Public.GO5_RobGrip1Status = 0;
   END_TRANSITION
   STEP DataMove_7:   // S270, max time T#10S, warning time T#7S
                   //"AutoProcessData_Buffer".DataBuffer["AutoProcessData".GlobalData.DataIndex]:="AutoProcessData".F_Robot3Grip2
                   //"AutoProcessData".GlobalData.DataIndex:="AutoProcessData".GlobalData.DataIndex+1
   END_STEP
   TRANSITION Trans271 FROM DataMove_7 TO "Data Clear_8"   // T271
      := #DataMove_7.T > t#100MS;
   END_TRANSITION

   // sequencer 15: S800-S859 ScanNG3 Put
   STEP "NG 3 PutProcess":   // S800, max time T#10S, warning time T#7S
   END_STEP
   TRANSITION Trans752 FROM "NG 3 PutProcess" TO StartRobotNG3Put   // T800
      := TRUE;
   END_TRANSITION
   STEP "Data Clear_9":   // S269, max time T#10S, warning time T#7S
              N    "AutoProcessData".F_Robot3Grip2:="AutoProcessData".ClearData
   END_STEP
   TRANSITION Trans270 FROM "Data Clear_9" TO WaitRobotFinish_11   // T270
      := TRUE;
   END_TRANSITION
   STEP StartRobotNG3Put:   // S376, max time T#10S, warning time T#7S
              N    "KukaRobot3_CtrlDB".sPLCtoROB.User.Cycle.DI267_LoadScanNGReq3
   END_STEP
   TRANSITION Trans653 FROM StartRobotNG3Put TO WaitRobotGripStatus_6   // T688
      := "KukaRobot3_CtrlDB".sROBtoPLC.User.Cycle.DO265_LoadNGInside AND NOT "KukaRobot3_CtrlDB".sROBtoPLC.User.Cycle.DO266_LoadNGFinish;
   END_TRANSITION
   STEP WaitRobotFinish_11:   // S377, max time T#10S, warning time T#7S
   END_STEP
   TRANSITION P19 FROM WaitRobotFinish_11 TO "NG3 PutProcessFinish"   // T689
      := "KukaRobot3_CtrlDB".sROBtoPLC.User.Cycle.DO266_LoadNGFinish;
   END_TRANSITION
   STEP "NG3 PutProcessFinish":   // S849, max time T#10S, warning time T#7S
              S    #ioPM_Inface.ProcessComplete
              R    #ioPM_Inface.ProcessStart
   END_STEP
   TRANSITION Trans682 FROM "NG3 PutProcessFinish" TO ProcessStart   // T849, jump
      := TRUE;
   END_TRANSITION
   STEP WaitRobotGripStatus_6:   // S378, max time T#10S, warning time T#7S
   END_STEP
   TRANSITION Trans683 FROM WaitRobotGripStatus_6 TO DataMove_8   // T690
      := "KukaRobot3_CtrlDB".sROBtoPLC.User.Public.GO6_RobGrip2Status = 0;
   END_TRANSITION
   STEP DataMove_8:   // S271, max time T#10S, warning time T#7S
                   //"AutoProcessData_Buffer".DataBuffer["AutoProcessData".GlobalData.DataIndex]:="AutoProcessData".F_Robot3Grip2
                   //"AutoProcessData".GlobalData.DataIndex:="AutoProcessData".GlobalData.DataIndex+1
   END_STEP
   TRANSITION Trans272 FROM DataMove_8 TO "Data Clear_9"   // T272
      := #DataMove_8.T > t#100MS;
   END_TRANSITION

   // sequencer 16: S850-S899 Maintenance Pos
   STEP "Maintenance Pos":   // S850, max time T#10S, warning time T#7S
   END_STEP
   TRANSITION Trans705 FROM "Maintenance Pos" TO ReqRobotToMantenPos_1   // T850
      := TRUE;
   END_TRANSITION
   STEP ReqRobotToMantenPos_1:   // S704, max time T#10S, warning time T#7S
              N    "KukaRobot3_CtrlDB".sPLCtoROB.User.Cycle.DI297_MaintainRequest
   END_STEP
   TRANSITION Trans706 FROM ReqRobotToMantenPos_1 TO WaitR1MaintenPosFinsh_1   // T705
      := "KukaRobot3_CtrlDB".sROBtoPLC.User.Cycle.DO297_MaintainInside AND NOT "KukaRobot3_CtrlDB".sROBtoPLC.User.Cycle.DO298_MaintainFinish;
   END_TRANSITION
   STEP WaitR1MaintenPosFinsh_1:   // S705, max time T#10S, warning time T#7S
              R    "AutoProcessControl".Robot_3.MaintenanceRequest
   END_STEP
   TRANSITION Trans707 FROM WaitR1MaintenPosFinsh_1 TO WaitRobotHomeRequest   // T706
      := NOT "KukaRobot3_CtrlDB".sROBtoPLC.User.Cycle.DO297_MaintainInside AND "KukaRobot3_CtrlDB".sROBtoPLC.User.Cycle.DO298_MaintainFinish AND NOT "AutoProcessControl".Robot_3.MaintenanceRequest AND NOT "ChangeOver_DB".Robot_3.Req_RobotToMaintenancePos;
   END_TRANSITION
   STEP WaitRobotHomeRequest:   // S706, max time T#10S, warning time T#7S
          S1  R    "ChangeOver_DB".Robot_3.MaintenancePosReqSelFlag
   END_STEP
   TRANSITION Trans708 FROM WaitRobotHomeRequest TO ReqRobotToHomePos   // T707
      := "AutoProcessControl".Robot_3.HomeRequest OR ("ChangeOver_DB".Robot_3.HMI_MaintenanceHomeReq AND NOT "KukaRobot3_CtrlDB".sROBtoPLC.User.Cycle.DO300_HomeInside);
   END_TRANSITION
   STEP ReqRobotToHomePos:   // S707, max time T#10S, warning time T#7S
              N    "KukaRobot3_CtrlDB".sPLCtoROB.User.Cycle.DI300_HomeRequest
   END_STEP
   TRANSITION Trans709 FROM ReqRobotToHomePos TO WaitR1HomePosFinsh_1   // T708
      := "KukaRobot3_CtrlDB".sROBtoPLC.User.Cycle.DO300_HomeInside AND NOT "KukaRobot3_CtrlDB".sROBtoPLC.User.Cycle.DO301_HomeFinish;
   END_TRANSITION
   STEP WaitR1HomePosFinsh_1:   // S899, max time T#10S, warning time T#7S
              R    "AutoProcessControl".Robot_3.HomeRequest
   END_STEP
   TRANSITION Trans712 FROM WaitR1HomePosFinsh_1 TO ProcessStart   // T899, jump
      := NOT "KukaRobot3_CtrlDB".sROBtoPLC.User.Cycle.DO300_HomeInside AND "KukaRobot3_CtrlDB".sROBtoPLC.User.Cycle.DO301_HomeFinish AND NOT "AutoProcessControl".Robot_3.HomeRequest;
   END_TRANSITION

   // sequencer 17: S900S950 Test
   STEP "900":   // S900, max time T#10S, warning time T#7S
   END_STEP
   TRANSITION Trans135 FROM "900" TO MasteringTest_Req   // T134
      := TRUE;
   END_TRANSITION
   TRANSITION Trans137 FROM "900" TO BrakeTest_Req   // T137
      := TRUE;
   END_TRANSITION
   STEP MasteringTest_Req:   // S910, max time T#10S, warning time T#7S
              N    "KukaRobot3_CtrlDB".sPLCtoROB.User.Cycle.DI321
              N    "KukaRobot3_CtrlDB".sPLCtoROB.User.Safety.DI450
   END_STEP
   TRANSITION Trans136 FROM MasteringTest_Req TO WaitMasteringTestFinish   // T136
      := "KukaRobot3_CtrlDB".sROBtoPLC.User.Safety.DO462;
   END_TRANSITION
   STEP BrakeTest_Req:   // S920, max time T#10S, warning time T#7S
              N    "KukaRobot3_CtrlDB".sPLCtoROB.User.Cycle.DI329
              N    "KukaRobot3_CtrlDB".sPLCtoROB.User.Safety.DI451
   END_STEP
   TRANSITION Trans138 FROM BrakeTest_Req TO WaitBrakeTestFinish   // T138
      := "KukaRobot3_CtrlDB".sROBtoPLC.User.Safety.DO453;
   END_TRANSITION
   STEP WaitMasteringTestFinish:   // S911, max time T#10S, warning time T#7S
   END_STEP
   TRANSITION Trans139 FROM WaitMasteringTestFinish TO MasteringTestFinish   // T139
      := NOT "KukaRobot3_CtrlDB".sROBtoPLC.User.Safety.DO460 AND NOT "KukaRobot3_CtrlDB".sROBtoPLC.User.Safety.DO462 AND "KukaRobot3_CtrlDB".sROBtoPLC.User.Safety.DO461;
   END_TRANSITION
   STEP WaitBrakeTestFinish:   // S921, max time T#10S, warning time T#7S
   END_STEP
   TRANSITION Trans141 FROM WaitBrakeTestFinish TO BrakeTestFinish   // T141
      := NOT "KukaRobot3_CtrlDB".sROBtoPLC.User.Safety.DO452 AND NOT "KukaRobot3_CtrlDB".sROBtoPLC.User.Safety.DO453 AND "KukaRobot3_CtrlDB".sROBtoPLC.User.Safety.DO454;
   END_TRANSITION
   STEP MasteringTestFinish:   // S919, max time T#10S, warning time T#7S
              R    "Robot_DB".Robot_3.MasteringTest_Req
   END_STEP
   TRANSITION Trans142 FROM MasteringTestFinish TO ProcessStart   // T919, jump
      := NOT "Robot_DB".Robot_3.MasteringTest_Req;
   END_TRANSITION
   STEP BrakeTestFinish:   // S929, max time T#10S, warning time T#7S
              R    "Robot_DB".Robot_3.BrakeTest_Req
   END_STEP
   TRANSITION Trans995 FROM BrakeTestFinish TO ProcessStart   // T929, jump
      := NOT "Robot_DB".Robot_3.BrakeTest_Req;
   END_TRANSITION

   // permanent post-instructions
   NETWORK 1
      #ioPM_Inface.StepNum := #RT_DATA.S_DISPLAY;
   NETWORK 2
      IF #iSysInface.Reset THEN #AlarmID := 0; END_IF;
   NETWORK 3
      #TON[10].TON(IN := #工件放行中, PT := T#0.5S);
      IF #TON[10].Q THEN #工件放行中 := FALSE; END_IF;
END_FUNCTION_BLOCK
